// TIA Portal V20 export
DATA_BLOCK "InstCallEquipment"   // DB135
{ DB_Accessible_From_OPC_UA := 'FALSE' }
AUTHOR : ERsystem_FA2_DH. Kim
// stored: AssignedProDiagFB Unit1.Em4.ProDiag, DBAccessibleFromOPCUA false, DBAccessibleFromWebserver false, InstanceOfName Unit1.Em4.CallEquipment, InstanceOfType FB, Namespace Unit1.Em4
"Unit1.Em4.CallEquipment"
   // VAR_INPUT
   //    ZoneOperationEnable { ExternalWritable := 'False'} : "LWONIK_typeSafetyZoneManualOperation";
   // END_VAR
   // VAR_IN_OUT
   //    unitStatus : "LAF_typeUnitStatus";
   //    unitAlarmDB : "LAF_typeAlarms";
   //    emFeedback : "LUC_typeEmFeedback";
   // END_VAR
   // VAR
   //    InstSequenceMainPnP : "Unit1.Em4.Sequence_1_MainPnP";
   //    InstSequenceAlignTable : "Unit1.Em4.Sequence_2_AlignTable";
   //    InstSequenceNgPnP : "Unit1.Em4.Sequence_3_NgPnP";
   //    InstSequenceGaugeRnR : "Unit1.Em4.Sequence_10_GaugeRnR";
   //    instMainPnPHomeJob1 : "LAF_SelectJob";
   //    instMainPnPHomeJob10 : "LAF_SelectJob";
   //    instMainPnPLoadJob2 : "LAF_SelectJob";
   //    instMainPnPUnloadJob3 : "LAF_SelectJob";
   //    instMainPnPAvoidJob4 : "LAF_SelectJob";
   //    instMainPnPOneLoadJob5 : "LAF_SelectJob";
   //    instMainPnPOneUnLoadJob6 : "LAF_SelectJob";
   //    instMainPnPDownWaitJob7 { S7_SetPoint := 'True'} : "LAF_SelectJob";
   //    instAlignTableHomeJob1 : "LAF_SelectJob";
   //    instAlignTableLoadJob2 : "LAF_SelectJob";
   //    instAlignTableVisionJob3 : "LAF_SelectJob";
   //    instAlignTableUnloadJob4 : "LAF_SelectJob";
   //    instAlignTableMotionJob22 : "LAF_SelectJob";
   //    instNgPnPHomeJob1 : "LAF_SelectJob";
   //    instNgPnPLoadJob2 : "LAF_SelectJob";
   //    instNgPnPUnloadJob3 : "LAF_SelectJob";
   //    instGaugeRnRCommonReadyJob1 : "LAF_SelectJob";
   //    instGaugeRnRCommonGetMasterPieceJob2 : "LAF_SelectJob";
   //    instGaugeRnRCommonMainPnPMoveAlignTableStackTableJob3 : "LAF_SelectJob";
   //    instGaugeRnRCommonMainPnp1ToAlignTableJob4 : "LAF_SelectJob";
   //    instGaugeRnRCommonMainPnPMoveReelCutConvyorAlignTableJob5 : "LAF_SelectJob";
   //    instGaugeRnRCommonAlignTableVisionAdjustJob6 : "LAF_SelectJob";
   //    instGaugeRnR1AlignAlignTableToMainPnP1Job10 { S7_SetPoint := 'True'} : "LAF_SelectJob";
   //    instGaugeRnR1AlignMainPnPMoveReelCutConvyorAlignTableJob11 { S7_SetPoint := 'True'} : "LAF_SelectJob";
   //    instGaugeRnR1AlignAlignTableMoveWaitJob12 { S7_SetPoint := 'True'} : "LAF_SelectJob";
   //    instGaugeRnR1AlignUnloadMasterPieceJob13 { S7_SetPoint := 'True'} : "LAF_SelectJob";
   //    instGaugeRnR1StackMainPnPMoveReelCutConvyorAlignTableJob15 { S7_SetPoint := 'True'} : "LAF_SelectJob";
   //    instGaugeRnR1StackAlignTableToMainPnP2Job16 { S7_SetPoint := 'True'} : "LAF_SelectJob";
   //    instGaugeRnR1StackMainPnPMoveAlignTableJob17 { S7_SetPoint := 'True'} : "LAF_SelectJob";
   //    instGaugeRnR1StackAlignTableMoveWaitJob18 { S7_SetPoint := 'True'} : "LAF_SelectJob";
   //    instGaugeRnR1StackMainPnP2ToStackTableJob19 { S7_SetPoint := 'True'} : "LAF_SelectJob";
   //    instGaugeRnR1StackStackTableToMainPnP2Job20 { S7_SetPoint := 'True'} : "LAF_SelectJob";
   //    instGaugeRnR1StackMainPnPMoveReelCutConvyorAlignTableJob21 { S7_SetPoint := 'True'} : "LAF_SelectJob";
   //    instGaugeRnR1StackMainPnP2ToAlignTableJob22 { S7_SetPoint := 'True'} : "LAF_SelectJob";
   //    instGaugeRnR1StackMainPnPMoveAlignTableJob23 { S7_SetPoint := 'True'} : "LAF_SelectJob";
   //    instGaugeRnR1StackAlignTableToMainPnP1Job24 { S7_SetPoint := 'True'} : "LAF_SelectJob";
   //    instGaugeRnR1StackMainPnPMoveReelCutConvyorAlignTableJob25 { S7_SetPoint := 'True'} : "LAF_SelectJob";
   //    instGaugeRnR1StackUnloadMasterPieceJob26 { S7_SetPoint := 'True'} : "LAF_SelectJob";
   //    instGaugeRnR3AlignMainPnPMoveReelCutConvyorAlignTableJob30 { S7_SetPoint := 'True'} : "LAF_SelectJob";
   //    instGaugeRnR3AlignNGPnPLoadMasterPieceJob31 { S7_SetPoint := 'True'} : "LAF_SelectJob";
   //    instGaugeRnR3AlignMainPnP2MoveAlignTableJob32 { S7_SetPoint := 'True'} : "LAF_SelectJob";
   //    instGaugeRnR3AlignAlignTableMoveWaitJob33 { S7_SetPoint := 'True'} : "LAF_SelectJob";
   //    instGaugeRnRCommonCheckCompleteJob39 { S7_SetPoint := 'True'} : "LAF_SelectJob";
   //    instCmPnp1stAnodeDetectSensor { S7_SetPoint := 'True'} : "LBC_DigitalSignalCn";
   //    instCmPnp2ndAnodeDetectSensor { S7_SetPoint := 'True'} : "LBC_DigitalSignalCn";
   //    instCmAnodeAlignTableElectrodeDetectSensor { S7_SetPoint := 'True'} : "LBC_DigitalSignalCn";
   //    instCmAnodeNgBoxFullSensorDetectSensor { S7_SetPoint := 'True'} : "LBC_DigitalSignalCn";
   //    instCmAnodeNgBoxDetectSensor { S7_SetPoint := 'True'} : "LBC_DigitalSignalCn";
   //    instCmAnodeMainPnP1AxisX { S7_SetPoint := 'True'} : "LBC_Axis64Pos_TecPlcCn";
   //    instCmAnodeMainPnP2AxisX { S7_SetPoint := 'True'} : "LBC_Axis64Pos_TecPlcCn";
   //    instCmAnodeMainPnP1AxisY { S7_SetPoint := 'True'} : "LBC_Axis64Pos_TecPlcCn";
   //    instCmAnodeMainPnP1AxisZ { S7_SetPoint := 'True'} : "LBC_Axis64Pos_TecPlcCn";
   //    instCmAnodeMainPnP2AxisZ { S7_SetPoint := 'True'} : "LBC_Axis64Pos_TecPlcCn";
   //    instCmAnodeAlignTableAxisX { S7_SetPoint := 'True'} : "LBC_Axis64Pos_TecPlcCn";
   //    instCmAnodeAlignTableAxisY1 { S7_SetPoint := 'True'} : "LBC_Axis64Pos_TecPlcCn";
   //    instCmAnodeAlignTableAxisY2 { S7_SetPoint := 'True'} : "LBC_Axis64Pos_TecPlcCn";
   //    instInterlockAnodeMainPnP1AxisX { S7_SetPoint := 'True'} : "LER_Axis64Pos_InterlockSummary";
   //    instInterlockAnodeMainPnP1AxisY { S7_SetPoint := 'True'} : "LER_Axis64Pos_InterlockSummary";
   //    instInterlockAnodeMainPnP1AxisZ { S7_SetPoint := 'True'} : "LER_Axis64Pos_InterlockSummary";
   //    instInterlockAnodeMainPnP2AxisX { S7_SetPoint := 'True'} : "LER_Axis64Pos_InterlockSummary";
   //    instInterlockAnodeMainPnP2AxisZ { S7_SetPoint := 'True'} : "LER_Axis64Pos_InterlockSummary";
   //    instInterlockAnodeAlignTableAxisX { S7_SetPoint := 'True'} : "LER_Axis64Pos_InterlockSummary";
   //    instInterlockAnodeAlignTableAxisY1 { S7_SetPoint := 'True'} : "LER_Axis64Pos_InterlockSummary";
   //    instInterlockAnodeAlignTableAxisY2 { S7_SetPoint := 'True'} : "LER_Axis64Pos_InterlockSummary";
   //    instAnodeMainPnP1AxisXSoftCam : "LER_SoftCam_Interface";
   //    instAnodeMainPnP2AxisXSoftCam { S7_SetPoint := 'True'} : "LER_SoftCam_Interface";
   //    instAnodeMainPnP1AxisYSoftCam { S7_SetPoint := 'True'} : "LER_SoftCam_Interface";
   //    instAnodeMainPnP1AxisZSoftCam { S7_SetPoint := 'True'} : "LER_SoftCam_Interface";
   //    instAnodeMainPnP2AxisZSoftCam { S7_SetPoint := 'True'} : "LER_SoftCam_Interface";
   //    instAnodeAlignTableAxisXSoftCam { S7_SetPoint := 'True'} : "LER_SoftCam_Interface";
   //    instAnodeAlignTableAxisY1SoftCam { S7_SetPoint := 'True'} : "LER_SoftCam_Interface";
   //    instAnodeAlignTableAxisY2SoftCam { S7_SetPoint := 'True'} : "LER_SoftCam_Interface";
   //    instCmAnodeMainPnP1RotaryCwCcw { ExternalAccessible := 'False'; ExternalVisible := 'False'; ExternalWritable := 'False'} : "LBC_TwoWayActuatorCn";
   //    instCmAnodeMainPnP1stSuctionPlateVacuum { ExternalAccessible := 'False'; ExternalVisible := 'False'; ExternalWritable := 'False'} : "LBC_TwoWayActuatorCn";
   //    instCmAnodeMainPnP2ndSuctionPlateVacuum { ExternalAccessible := 'False'; ExternalVisible := 'False'; ExternalWritable := 'False'} : "LBC_TwoWayActuatorCn";
   //    instCmAnodeAlignTableSuctionPlateVacuum { ExternalAccessible := 'False'; ExternalVisible := 'False'; ExternalWritable := 'False'; S7_SetPoint := 'True'} : "LBC_TwoWayActuatorCn";
   //    instCmAnodeGlassCleaning { ExternalAccessible := 'False'; ExternalVisible := 'False'; ExternalWritable := 'False'; S7_SetPoint := 'True'} : "LBC_TwoWayActuatorCn";
   //    instCmAnodeNgPnpUpDown { ExternalAccessible := 'False'; ExternalVisible := 'False'; ExternalWritable := 'False'; S7_SetPoint := 'True'} : "LBC_TwoWayActuatorCn";
   //    instCmAnodeNgPnp1stFwdBwd { ExternalAccessible := 'False'; ExternalVisible := 'False'; ExternalWritable := 'False'; S7_SetPoint := 'True'} : "LBC_TwoWayActuatorCn";
   //    instCmAnodeNgPnp2ndFwdBwd { ExternalAccessible := 'False'; ExternalVisible := 'False'; ExternalWritable := 'False'; S7_SetPoint := 'True'} : "LBC_TwoWayActuatorCn";
   //    instCmAnodeMaintenanceMovingFixFwdBwd { ExternalAccessible := 'False'; ExternalVisible := 'False'; ExternalWritable := 'False'; S7_SetPoint := 'True'} : "LBC_TwoWayActuatorCn";
   //    instCmAnodeNgBoxLiftUpDown { ExternalAccessible := 'False'; ExternalVisible := 'False'; ExternalWritable := 'False'; S7_SetPoint := 'True'} : "LBC_TwoWayActuatorCn";
   //    instCmAnodeNgBoxLockUpDown { ExternalAccessible := 'False'; ExternalVisible := 'False'; ExternalWritable := 'False'; S7_SetPoint := 'True'} : "LBC_TwoWayActuatorCn";
   //    instCmAnodeNgPnpVaccum { ExternalAccessible := 'False'; ExternalVisible := 'False'; ExternalWritable := 'False'; S7_SetPoint := 'True'} : "LBC_TwoWayActuatorCn";
   //    instCmAnodeConveyorCoverFwdBwd { S7_SetPoint := 'True'} : "LBC_TwoWayActuatorCn";
   //    instCmAnodeConveyorPickUpBlower { S7_SetPoint := 'True'} : "LBC_TwoWayActuatorCn";
   //    instCmAnodeVisionControllerInterface { ExternalAccessible := 'False'; ExternalVisible := 'False'; ExternalWritable := 'False'; S7_SetPoint := 'True'} : "LER_Vision_XGX2000";
   //    instAlignVisionConversion : "LER_AlignVisionConversion";
   //    instManageAlarms { ExternalWritable := 'False'} : "LAF_ManageAlarms";
   //    instLER_BrakeTestAnodeMainPnP1AxisZ : "LER_BrakeTest";
   //    instLER_BrakeTestAnodeMainPnP2AxisZ { S7_SetPoint := 'True'} : "LER_BrakeTest";
   //    instEventsPFE : "Unit1.Em4.EventsPFE";
   //    statUnitStatus { ExternalWritable := 'False'} : "LAF_typeUnitStatus";
   //    statSlmStatus { ExternalWritable := 'False'} : Struct
   //       running : Bool;
   //       powerOff : Bool;
   //    END_STRUCT;
   //    statAllBrakeTest { ExternalWritable := 'False'} : "LER_typeBrakeTestUnitCommands";
   //    statInterlockTonTime { ExternalAccessible := 'False'; ExternalVisible := 'False'; ExternalWritable := 'False'} : Struct
   //       mainPnP1AxisX : Array[0..15] of TON_TIME;
   //       mainPnP1AxisY : Array[0..15] of TON_TIME;
   //       mainPnP1AxisZ : Array[0..15] of TON_TIME;
   //       mainPnP2AxisX : Array[0..15] of TON_TIME;
   //       mainPnP2AxisZ : Array[0..15] of TON_TIME;
   //       alignTableAxisX : Array[0..15] of TON_TIME;
   //       alignTableAxisY1 : Array[0..15] of TON_TIME;
   //       alignTableAxisY2 : Array[0..15] of TON_TIME;
   //    END_STRUCT;
   //    statTonTime { ExternalAccessible := 'False'; ExternalVisible := 'False'; ExternalWritable := 'False'} : Array[0..1999] of TON_TIME;
   //    statTofTime { ExternalAccessible := 'False'; ExternalVisible := 'False'; ExternalWritable := 'False'} : Array[0..99] of TOF_TIME;
   //    statPulse { ExternalAccessible := 'False'; ExternalVisible := 'False'; ExternalWritable := 'False'} : Struct
   //       miscellaneous : Array[0..99] of Bool;
   //       workingDone : Struct
   //          mainPnP : Array[0..99] of Bool;
   //          alignTable : Array[0..99] of Bool;
   //          ngPnP : Array[0..99] of Bool;
   //       END_STRUCT;
   //       axisEnable : Array[0..99] of Bool;
   //       brakeTest : Array[0..99] of Bool;
   //    END_STRUCT;
   //    statEnableManualCmds : Bool := TRUE;
   //    Scan_on : Bool;
   //    "*** Interlock Axis ***" { ExternalAccessible := 'False'; ExternalVisible := 'False'; ExternalWritable := 'False'} : Bool;
   //    "AnodeMainPnP1AxisX Home" { S7_SetPoint := 'True'} : "Homing.LER_Axis";
   //    "AnodeMainPnP1AxisX Jog_CW" { S7_SetPoint := 'True'} : "Jog.LER_Axis";
   //    "AnodeMainPnP1AxisX Jog_CCW" { S7_SetPoint := 'True'} : "Jog.LER_Axis";
   //    "AnodeMainPnP1AxisX Position_" { S7_SetPoint := 'True'} : Array[0..5] of "Position.LER_Axis";
   //    "AnodeMainPnP2AxisX Home" { S7_SetPoint := 'True'} : "Homing.LER_Axis";
   //    "AnodeMainPnP2AxisX Jog_CW" { S7_SetPoint := 'True'} : "Jog.LER_Axis";
   //    "AnodeMainPnP2AxisX Jog_CCW" { S7_SetPoint := 'True'} : "Jog.LER_Axis";
   //    "AnodeMainPnP2AxisX Position_" { S7_SetPoint := 'True'} : Array[0..5] of "Position.LER_Axis";
   //    "AnodeMainPnP1AxisY Home" { S7_SetPoint := 'True'} : "Homing.LER_Axis";
   //    "AnodeMainPnP1AxisY Jog_CW" { S7_SetPoint := 'True'} : "Jog.LER_Axis";
   //    "AnodeMainPnP1AxisY Jog_CCW" { S7_SetPoint := 'True'} : "Jog.LER_Axis";
   //    "AnodeMainPnP1AxisY Position_" { S7_SetPoint := 'True'} : Array[0..5] of "Position.LER_Axis";
   //    "AnodeMainPnP1AxisZ Home" { S7_SetPoint := 'True'} : "Homing.LER_Axis";
   //    "AnodeMainPnP1AxisZ Jog_CW" { S7_SetPoint := 'True'} : "Jog.LER_Axis";
   //    "AnodeMainPnP1AxisZ Jog_CCW" { S7_SetPoint := 'True'} : "Jog.LER_Axis";
   //    "AnodeMainPnP1AxisZ Position_" { S7_SetPoint := 'True'} : Array[0..5] of "Position.LER_Axis";
   //    "AnodeMainPnP2AxisZ Home" { S7_SetPoint := 'True'} : "Homing.LER_Axis";
   //    "AnodeMainPnP2AxisZ Jog_CW" { S7_SetPoint := 'True'} : "Jog.LER_Axis";
   //    "AnodeMainPnP2AxisZ Jog_CCW" { S7_SetPoint := 'True'} : "Jog.LER_Axis";
   //    "AnodeMainPnP2AxisZ Position_" { S7_SetPoint := 'True'} : Array[0..5] of "Position.LER_Axis";
   //    "AnodeAlignTableAxisX Home" { S7_SetPoint := 'True'} : "Homing.LER_Axis";
   //    "AnodeAlignTableAxisX Jog_CW" { S7_SetPoint := 'True'} : "Jog.LER_Axis";
   //    "AnodeAlignTableAxisX Jog_CCW" { S7_SetPoint := 'True'} : "Jog.LER_Axis";
   //    "AnodeAlignTableAxisX Position_" { S7_SetPoint := 'True'} : Array[0..5] of "Position.LER_Axis";
   //    "AnodeAlignTableAxisY1 Home" { S7_SetPoint := 'True'} : "Homing.LER_Axis";
   //    "AnodeAlignTableAxisY1 Jog_CW" { S7_SetPoint := 'True'} : "Jog.LER_Axis";
   //    "AnodeAlignTableAxisY1 Jog_CCW" { S7_SetPoint := 'True'} : "Jog.LER_Axis";
   //    "AnodeAlignTableAxisY1 Position_" { S7_SetPoint := 'True'} : Array[0..5] of "Position.LER_Axis";
   //    "AnodeAlignTableAxisY2 Home" { S7_SetPoint := 'True'} : "Homing.LER_Axis";
   //    "AnodeAlignTableAxisY2 Jog_CW" { S7_SetPoint := 'True'} : "Jog.LER_Axis";
   //    "AnodeAlignTableAxisY2 Jog_CCW" { S7_SetPoint := 'True'} : "Jog.LER_Axis";
   //    "AnodeAlignTableAxisY2 Position_" { S7_SetPoint := 'True'} : Array[0..5] of "Position.LER_Axis";
   //    "*** Interlock Actuator ******" { ExternalAccessible := 'False'; ExternalVisible := 'False'; ExternalWritable := 'False'} : Bool;
   //    "AnodeNgBoxLiftUpDown Home" { S7_SetPoint := 'True'} : "Cylinder.LER_Actuator";
   //    "AnodeNgBoxLiftUpDown Work" { S7_SetPoint := 'True'} : "Cylinder.LER_Actuator";
   //    "AnodeNgBoxLockUpDown Home" { S7_SetPoint := 'True'} : "Cylinder.LER_Actuator";
   //    "AnodeNgBoxLockUpDown Work" { S7_SetPoint := 'True'} : "Cylinder.LER_Actuator";
   //    "AnodeMaintenanceMovingFixFrontFwdBwd Home" { S7_SetPoint := 'True'} : "Cylinder.LER_Actuator";
   //    "AnodeMaintenanceMovingFixFrontFwdBwd Work" { S7_SetPoint := 'True'} : "Cylinder.LER_Actuator";
   //    "AnodeGlassCleaning Home" { S7_SetPoint := 'True'} : "Cylinder.LER_Actuator";
   //    "AnodeGlassCleaning Work" { S7_SetPoint := 'True'} : "Cylinder.LER_Actuator";
   //    "AnodeNgPnp1stFwdBwd Home" { S7_SetPoint := 'True'} : "Cylinder.LER_Actuator";
   //    "AnodeNgPnp1stFwdBwd Work" { S7_SetPoint := 'True'} : "Cylinder.LER_Actuator";
   //    "AnodeNgPnpUpDown Home" { S7_SetPoint := 'True'} : "Cylinder.LER_Actuator";
   //    "AnodeNgPnpUpDown Work" { S7_SetPoint := 'True'} : "Cylinder.LER_Actuator";
   //    "AnodeMainPnP1RotaryCwCcw Home" { S7_SetPoint := 'True'} : "Cylinder.LER_Actuator";
   //    "AnodeMainPnP1RotaryCwCcw Work" { S7_SetPoint := 'True'} : "Cylinder.LER_Actuator";
   //    "AnodeNgPnp2ndFwdBwd Home" { S7_SetPoint := 'True'} : "Cylinder.LER_Actuator";
   //    "AnodeNgPnp2ndFwdBwd Work" { S7_SetPoint := 'True'} : "Cylinder.LER_Actuator";
   //    Tracking_04 { S7_SetPoint := 'True'} : "Unit1.Em4.PartData";
   //    AXIS5 : "LER_CM_Name";
   //    AXIS11 : "LER_CM_Name";
   //    AXIS14 : "LER_CM_Name";
   //    Cylinder13 : "LER_CM_Name";
   //    Cylinder18 : "LER_CM_Name";
   //    Vaccum10 : "LER_CM_Name";
   //    instAlignVisionHistory { S7_SetPoint := 'True'} : "LER_visionHistory";
   //    instAlignMoveCalibration { S7_SetPoint := 'True'} : "LER_AlignMoveCalibration";
   //    instAlignThetaCalibration { S7_SetPoint := 'True'} : "LER_AlignThetaCalibration";
   //    instAlignSyncMove { S7_SetPoint := 'True'} : "LER_AlignSyncMove";
   //    citi_Ptrig : Array[0..20] of Bool;
   //    citiTon : Array[0..20] of TON_TIME;
   //    citi : Time;
   //    citiTest : Array[0..20] of Bool;
   // END_VAR
BEGIN
   ZoneOperationEnable.autoStartEnable := FALSE;
   ZoneOperationEnable.doorLockEnable := TRUE;
   ZoneOperationEnable.doorUnlockEnable := TRUE;
   ZoneOperationEnable.rc_AutoEnable := FALSE;
   ZoneOperationEnable.rc_RollChangeEnable := FALSE;
   ZoneOperationEnable.rc_DoorLockEnable := TRUE;
   ZoneOperationEnable.rc_DoorUnlockEnable := TRUE;
   ZoneOperationEnable.hmiOperationEnable := TRUE;
   ZoneOperationEnable.phmiOperationEnable := FALSE;
   instCmPnp1stAnodeDetectSensor.enable := TRUE;
   instCmPnp1stAnodeDetectSensor.parentReferenceDesignator := WSTRING#'';
   instCmPnp1stAnodeDetectSensor.digitalValue := FALSE;
   instCmPnp1stAnodeDetectSensor.simulatedDigitalValue := FALSE;
   instCmPnp1stAnodeDetectSensor.statProcessValues.enable := TRUE;
   instCmPnp1stAnodeDetectSensor.statProcessValues.referenceDesignator := WSTRING#'Pnp1stAnodeDetect';
   instCmPnp1stAnodeDetectSensor.statProcessValues.simulation := FALSE;
   instCmPnp1stAnodeDetectSensor.statProcessValues.processValue := FALSE;
   instCmPnp1stAnodeDetectSensor.statProcessValues.error := FALSE;
   instCmPnp1stAnodeDetectSensor.statProcessValues.status := 16#0000;
   instCmPnp1stAnodeDetectSensor.statDiagnostics.status := 16#0000;
   instCmPnp1stAnodeDetectSensor.statDiagnostics.subfunctionStatus := 16#0000;
   instCmPnp1stAnodeDetectSensor.statDiagnostics.stateNumber := 0;
   instCmPnp1stAnodeDetectSensor.statEmptyDiagnostics.status := 16#0000;
   instCmPnp1stAnodeDetectSensor.statEmptyDiagnostics.subfunctionStatus := 16#0000;
   instCmPnp1stAnodeDetectSensor.statEmptyDiagnostics.stateNumber := 0;
   instCmPnp1stAnodeDetectSensor.instOnDelay.PT := T#0MS;
   instCmPnp1stAnodeDetectSensor.instOnDelay.IN := FALSE;
   instCmPnp1stAnodeDetectSensor.instOffDelay.PT := T#0MS;
   instCmPnp1stAnodeDetectSensor.instOffDelay.IN := FALSE;
   instCmPnp1stAnodeDetectSensor.statDisableAlarms := FALSE;
   instCmPnp1stAnodeDetectSensor.statErrorState := 16#0000;
   instCmPnp1stAnodeDetectSensor.statFirstCall := FALSE;
   instCmPnp1stAnodeDetectSensor.statResetPrevious := FALSE;
   instCmPnp1stAnodeDetectSensor.statEnablePrevious := TRUE;
   instCmPnp1stAnodeDetectSensor.statProcessValuePrevious := FALSE;
   instCmPnp2ndAnodeDetectSensor.enable := TRUE;
   instCmPnp2ndAnodeDetectSensor.parentReferenceDesignator := WSTRING#'';
   instCmPnp2ndAnodeDetectSensor.digitalValue := FALSE;
   instCmPnp2ndAnodeDetectSensor.simulatedDigitalValue := FALSE;
   instCmPnp2ndAnodeDetectSensor.statProcessValues.enable := TRUE;
   instCmPnp2ndAnodeDetectSensor.statProcessValues.referenceDesignator := WSTRING#'Pnp2ndAnodeDetect';
   instCmPnp2ndAnodeDetectSensor.statProcessValues.simulation := FALSE;
   instCmPnp2ndAnodeDetectSensor.statProcessValues.processValue := FALSE;
   instCmPnp2ndAnodeDetectSensor.statProcessValues.error := FALSE;
   instCmPnp2ndAnodeDetectSensor.statProcessValues.status := 16#0000;
   instCmPnp2ndAnodeDetectSensor.statDiagnostics.status := 16#0000;
   instCmPnp2ndAnodeDetectSensor.statDiagnostics.subfunctionStatus := 16#0000;
   instCmPnp2ndAnodeDetectSensor.statDiagnostics.stateNumber := 0;
   instCmPnp2ndAnodeDetectSensor.statEmptyDiagnostics.status := 16#0000;
   instCmPnp2ndAnodeDetectSensor.statEmptyDiagnostics.subfunctionStatus := 16#0000;
   instCmPnp2ndAnodeDetectSensor.statEmptyDiagnostics.stateNumber := 0;
   instCmPnp2ndAnodeDetectSensor.instOnDelay.PT := T#0MS;
   instCmPnp2ndAnodeDetectSensor.instOnDelay.IN := FALSE;
   instCmPnp2ndAnodeDetectSensor.instOffDelay.PT := T#0MS;
   instCmPnp2ndAnodeDetectSensor.instOffDelay.IN := FALSE;
   instCmPnp2ndAnodeDetectSensor.statDisableAlarms := FALSE;
   instCmPnp2ndAnodeDetectSensor.statErrorState := 16#0000;
   instCmPnp2ndAnodeDetectSensor.statFirstCall := FALSE;
   instCmPnp2ndAnodeDetectSensor.statResetPrevious := FALSE;
   instCmPnp2ndAnodeDetectSensor.statEnablePrevious := TRUE;
   instCmPnp2ndAnodeDetectSensor.statProcessValuePrevious := FALSE;
   instCmAnodeAlignTableElectrodeDetectSensor.enable := TRUE;
   instCmAnodeAlignTableElectrodeDetectSensor.parentReferenceDesignator := WSTRING#'';
   instCmAnodeAlignTableElectrodeDetectSensor.digitalValue := FALSE;
   instCmAnodeAlignTableElectrodeDetectSensor.simulatedDigitalValue := FALSE;
   instCmAnodeAlignTableElectrodeDetectSensor.statProcessValues.enable := TRUE;
   instCmAnodeAlignTableElectrodeDetectSensor.statProcessValues.referenceDesignator := WSTRING#'AlignTableElectrodeDetect';
   instCmAnodeAlignTableElectrodeDetectSensor.statProcessValues.simulation := FALSE;
   instCmAnodeAlignTableElectrodeDetectSensor.statProcessValues.processValue := FALSE;
   instCmAnodeAlignTableElectrodeDetectSensor.statProcessValues.error := FALSE;
   instCmAnodeAlignTableElectrodeDetectSensor.statProcessValues.status := 16#0000;
   instCmAnodeAlignTableElectrodeDetectSensor.statDiagnostics.status := 16#0000;
   instCmAnodeAlignTableElectrodeDetectSensor.statDiagnostics.subfunctionStatus := 16#0000;
   instCmAnodeAlignTableElectrodeDetectSensor.statDiagnostics.stateNumber := 0;
   instCmAnodeAlignTableElectrodeDetectSensor.statEmptyDiagnostics.status := 16#0000;
   instCmAnodeAlignTableElectrodeDetectSensor.statEmptyDiagnostics.subfunctionStatus := 16#0000;
   instCmAnodeAlignTableElectrodeDetectSensor.statEmptyDiagnostics.stateNumber := 0;
   instCmAnodeAlignTableElectrodeDetectSensor.instOnDelay.PT := T#0MS;
   instCmAnodeAlignTableElectrodeDetectSensor.instOnDelay.IN := FALSE;
   instCmAnodeAlignTableElectrodeDetectSensor.instOffDelay.PT := T#0MS;
   instCmAnodeAlignTableElectrodeDetectSensor.instOffDelay.IN := FALSE;
   instCmAnodeAlignTableElectrodeDetectSensor.statDisableAlarms := FALSE;
   instCmAnodeAlignTableElectrodeDetectSensor.statErrorState := 16#0000;
   instCmAnodeAlignTableElectrodeDetectSensor.statFirstCall := FALSE;
   instCmAnodeAlignTableElectrodeDetectSensor.statResetPrevious := FALSE;
   instCmAnodeAlignTableElectrodeDetectSensor.statEnablePrevious := TRUE;
   instCmAnodeAlignTableElectrodeDetectSensor.statProcessValuePrevious := FALSE;
   instCmAnodeNgBoxFullSensorDetectSensor.enable := TRUE;
   instCmAnodeNgBoxFullSensorDetectSensor.parentReferenceDesignator := WSTRING#'';
   instCmAnodeNgBoxFullSensorDetectSensor.digitalValue := TRUE;
   instCmAnodeNgBoxFullSensorDetectSensor.simulatedDigitalValue := FALSE;
   instCmAnodeNgBoxFullSensorDetectSensor.statProcessValues.enable := TRUE;
   instCmAnodeNgBoxFullSensorDetectSensor.statProcessValues.referenceDesignator := WSTRING#'NgBoxFullSensorDetect';
   instCmAnodeNgBoxFullSensorDetectSensor.statProcessValues.simulation := FALSE;
   instCmAnodeNgBoxFullSensorDetectSensor.statProcessValues.processValue := TRUE;
   instCmAnodeNgBoxFullSensorDetectSensor.statProcessValues.error := FALSE;
   instCmAnodeNgBoxFullSensorDetectSensor.statProcessValues.status := 16#0000;
   instCmAnodeNgBoxFullSensorDetectSensor.statDiagnostics.status := 16#0000;
   instCmAnodeNgBoxFullSensorDetectSensor.statDiagnostics.subfunctionStatus := 16#0000;
   instCmAnodeNgBoxFullSensorDetectSensor.statDiagnostics.stateNumber := 0;
   instCmAnodeNgBoxFullSensorDetectSensor.statEmptyDiagnostics.status := 16#0000;
   instCmAnodeNgBoxFullSensorDetectSensor.statEmptyDiagnostics.subfunctionStatus := 16#0000;
   instCmAnodeNgBoxFullSensorDetectSensor.statEmptyDiagnostics.stateNumber := 0;
   instCmAnodeNgBoxFullSensorDetectSensor.instOnDelay.PT := T#0MS;
   instCmAnodeNgBoxFullSensorDetectSensor.instOnDelay.IN := FALSE;
   instCmAnodeNgBoxFullSensorDetectSensor.instOffDelay.PT := T#0MS;
   instCmAnodeNgBoxFullSensorDetectSensor.instOffDelay.IN := FALSE;
   instCmAnodeNgBoxFullSensorDetectSensor.statDisableAlarms := FALSE;
   instCmAnodeNgBoxFullSensorDetectSensor.statErrorState := 16#0000;
   instCmAnodeNgBoxFullSensorDetectSensor.statFirstCall := FALSE;
   instCmAnodeNgBoxFullSensorDetectSensor.statResetPrevious := FALSE;
   instCmAnodeNgBoxFullSensorDetectSensor.statEnablePrevious := TRUE;
   instCmAnodeNgBoxFullSensorDetectSensor.statProcessValuePrevious := TRUE;
   instCmAnodeNgBoxDetectSensor.enable := TRUE;
   instCmAnodeNgBoxDetectSensor.parentReferenceDesignator := WSTRING#'';
   instCmAnodeNgBoxDetectSensor.digitalValue := TRUE;
   instCmAnodeNgBoxDetectSensor.simulatedDigitalValue := FALSE;
   instCmAnodeNgBoxDetectSensor.statProcessValues.enable := TRUE;
   instCmAnodeNgBoxDetectSensor.statProcessValues.referenceDesignator := WSTRING#'NgBoxDetect';
   instCmAnodeNgBoxDetectSensor.statProcessValues.simulation := FALSE;
   instCmAnodeNgBoxDetectSensor.statProcessValues.processValue := TRUE;
   instCmAnodeNgBoxDetectSensor.statProcessValues.error := FALSE;
   instCmAnodeNgBoxDetectSensor.statProcessValues.status := 16#0000;
   instCmAnodeNgBoxDetectSensor.statDiagnostics.status := 16#0000;
   instCmAnodeNgBoxDetectSensor.statDiagnostics.subfunctionStatus := 16#0000;
   instCmAnodeNgBoxDetectSensor.statDiagnostics.stateNumber := 0;
   instCmAnodeNgBoxDetectSensor.statEmptyDiagnostics.status := 16#0000;
   instCmAnodeNgBoxDetectSensor.statEmptyDiagnostics.subfunctionStatus := 16#0000;
   instCmAnodeNgBoxDetectSensor.statEmptyDiagnostics.stateNumber := 0;
   instCmAnodeNgBoxDetectSensor.instOnDelay.PT := T#0MS;
   instCmAnodeNgBoxDetectSensor.instOnDelay.IN := FALSE;
   instCmAnodeNgBoxDetectSensor.instOffDelay.PT := T#0MS;
   instCmAnodeNgBoxDetectSensor.instOffDelay.IN := FALSE;
   instCmAnodeNgBoxDetectSensor.statDisableAlarms := FALSE;
   instCmAnodeNgBoxDetectSensor.statErrorState := 16#0000;
   instCmAnodeNgBoxDetectSensor.statFirstCall := FALSE;
   instCmAnodeNgBoxDetectSensor.statResetPrevious := FALSE;
   instCmAnodeNgBoxDetectSensor.statEnablePrevious := TRUE;
   instCmAnodeNgBoxDetectSensor.statProcessValuePrevious := TRUE;
   instCmAnodeMainPnP1RotaryCwCcw.enable := TRUE;
   instCmAnodeMainPnP1RotaryCwCcw.parentReferenceDesignator := WSTRING#'';
   instCmAnodeMainPnP1RotaryCwCcw.feedbackHomePos := FALSE;
   instCmAnodeMainPnP1RotaryCwCcw.feedbackWorkPos := TRUE;
   instCmAnodeMainPnP1RotaryCwCcw.enableManualCmds := TRUE;
   instCmAnodeMainPnP1RotaryCwCcw.interlockWorkPos := FALSE;
   instCmAnodeMainPnP1RotaryCwCcw.interlockHomePos := FALSE;
   instCmAnodeMainPnP1RotaryCwCcw.goToHomePos := FALSE;
   instCmAnodeMainPnP1RotaryCwCcw.goToWorkPos := FALSE;
   instCmAnodeMainPnP1RotaryCwCcw.statProcessValues.enable := TRUE;
   instCmAnodeMainPnP1RotaryCwCcw.statProcessValues.referenceDesignator := WSTRING#'MainPnP1RotaryCwCcw';
   instCmAnodeMainPnP1RotaryCwCcw.statProcessValues.commandHomePos := FALSE;
   instCmAnodeMainPnP1RotaryCwCcw.statProcessValues.commandWorkPos := FALSE;
   instCmAnodeMainPnP1RotaryCwCcw.statProcessValues.goToHomePos := FALSE;
   instCmAnodeMainPnP1RotaryCwCcw.statProcessValues.goToWorkPos := FALSE;
   instCmAnodeMainPnP1RotaryCwCcw.statProcessValues.inHomePos := FALSE;
   instCmAnodeMainPnP1RotaryCwCcw.statProcessValues.inWorkPos := FALSE;
   instCmAnodeMainPnP1RotaryCwCcw.statProcessValues.reset := FALSE;
   instCmAnodeMainPnP1RotaryCwCcw.statProcessValues.enableManualCmds := TRUE;
   instCmAnodeMainPnP1RotaryCwCcw.statProcessValues.error := FALSE;
   instCmAnodeMainPnP1RotaryCwCcw.statProcessValues.interlockHomePos := FALSE;
   instCmAnodeMainPnP1RotaryCwCcw.statProcessValues.interlockWorkPos := FALSE;
   instCmAnodeMainPnP1RotaryCwCcw.statProcessValues.status := 16#7100;
   instCmAnodeMainPnP1RotaryCwCcw.statProcessValues.interlockWarningWorkPos := FALSE;
   instCmAnodeMainPnP1RotaryCwCcw.statProcessValues.interlockWarningHomePos := FALSE;
   instCmAnodeMainPnP1RotaryCwCcw.statCurrentInputs.commandHomePos := FALSE;
   instCmAnodeMainPnP1RotaryCwCcw.statCurrentInputs.commandWorkPos := FALSE;
   instCmAnodeMainPnP1RotaryCwCcw.statCurrentInputs.reset := FALSE;
   instCmAnodeMainPnP1RotaryCwCcw.statPreviousInputs.commandHomePos := FALSE;
   instCmAnodeMainPnP1RotaryCwCcw.statPreviousInputs.commandWorkPos := FALSE;
   instCmAnodeMainPnP1RotaryCwCcw.statPreviousInputs.reset := FALSE;
   instCmAnodeMainPnP1RotaryCwCcw.statCurrentInterface.commandHomePos := FALSE;
   instCmAnodeMainPnP1RotaryCwCcw.statCurrentInterface.commandWorkPos := FALSE;
   instCmAnodeMainPnP1RotaryCwCcw.statCurrentInterface.reset := FALSE;
   instCmAnodeMainPnP1RotaryCwCcw.statPreviousInterface.commandHomePos := FALSE;
   instCmAnodeMainPnP1RotaryCwCcw.statPreviousInterface.commandWorkPos := FALSE;
   instCmAnodeMainPnP1RotaryCwCcw.statPreviousInterface.reset := FALSE;
   instCmAnodeMainPnP1RotaryCwCcw.statEmptyDiagnostics.status := 16#0000;
   instCmAnodeMainPnP1RotaryCwCcw.statEmptyDiagnostics.subfunctionStatus := 16#0000;
   instCmAnodeMainPnP1RotaryCwCcw.statEmptyDiagnostics.stateNumber := 0;
   instCmAnodeMainPnP1RotaryCwCcw.instTimerReachPos.PT := T#0MS;
   instCmAnodeMainPnP1RotaryCwCcw.instTimerReachPos.IN := FALSE;
   instCmAnodeMainPnP1RotaryCwCcw.instTimerLeavePos.PT := T#0MS;
   instCmAnodeMainPnP1RotaryCwCcw.instTimerLeavePos.IN := FALSE;
   instCmAnodeMainPnP1RotaryCwCcw.instTimerDiscrepancyCheck.PT := T#0MS;
   instCmAnodeMainPnP1RotaryCwCcw.instTimerDiscrepancyCheck.IN := FALSE;
   instCmAnodeMainPnP1RotaryCwCcw.statDisableAlarms := TRUE;
   instCmAnodeMainPnP1RotaryCwCcw.statDiagnostics.status := 16#7003;
   instCmAnodeMainPnP1RotaryCwCcw.statDiagnostics.subfunctionStatus := 16#0000;
   instCmAnodeMainPnP1RotaryCwCcw.statDiagnostics.stateNumber := 0;
   instCmAnodeMainPnP1RotaryCwCcw.statEnablePrevious := TRUE;
   instCmAnodeMainPnP1RotaryCwCcw.statFirstCall := FALSE;
   instCmAnodeMainPnP1RotaryCwCcw.statResetPrevious := FALSE;
   instCmAnodeMainPnP1RotaryCwCcw.statValid := TRUE;
   instCmAnodeMainPnP1RotaryCwCcw.statBusy := TRUE;
   instCmAnodeMainPnP1RotaryCwCcw.statError := FALSE;
   instCmAnodeMainPnP1RotaryCwCcw.statInterlockWorkOff := FALSE;
   instCmAnodeMainPnP1RotaryCwCcw.statInterlockHomeOff := FALSE;
   instCmAnodeMainPnP1RotaryCwCcw.statFbState := 50;
   instCmAnodeMainPnP1RotaryCwCcw.statFbStatePrevious := 50;
   instCmAnodeMainPnP1RotaryCwCcw.statErrorUserCleared := FALSE;
   instCmAnodeMainPnP1RotaryCwCcw.statErrorAutoCleared := FALSE;
   instCmAnodeMainPnP1RotaryCwCcw.statErrorState := 16#0000;
   instCmAnodeMainPnP1RotaryCwCcw.statDisablingCompleted := FALSE;
   instCmAnodeMainPnP1RotaryCwCcw.statFeedbackHomePos := FALSE;
   instCmAnodeMainPnP1RotaryCwCcw.statFeedbackWorkPos := TRUE;
   instCmAnodeMainPnP1stSuctionPlateVacuum.enable := TRUE;
   instCmAnodeMainPnP1stSuctionPlateVacuum.parentReferenceDesignator := WSTRING#'';
   instCmAnodeMainPnP1stSuctionPlateVacuum.feedbackHomePos := TRUE;
   instCmAnodeMainPnP1stSuctionPlateVacuum.feedbackWorkPos := FALSE;
   instCmAnodeMainPnP1stSuctionPlateVacuum.enableManualCmds := TRUE;
   instCmAnodeMainPnP1stSuctionPlateVacuum.interlockWorkPos := TRUE;
   instCmAnodeMainPnP1stSuctionPlateVacuum.interlockHomePos := TRUE;
   instCmAnodeMainPnP1stSuctionPlateVacuum.goToHomePos := FALSE;
   instCmAnodeMainPnP1stSuctionPlateVacuum.goToWorkPos := FALSE;
   instCmAnodeMainPnP1stSuctionPlateVacuum.statProcessValues.enable := TRUE;
   instCmAnodeMainPnP1stSuctionPlateVacuum.statProcessValues.referenceDesignator := WSTRING#'MainPnP1Vacuum';
   instCmAnodeMainPnP1stSuctionPlateVacuum.statProcessValues.commandHomePos := FALSE;
   instCmAnodeMainPnP1stSuctionPlateVacuum.statProcessValues.commandWorkPos := FALSE;
   instCmAnodeMainPnP1stSuctionPlateVacuum.statProcessValues.goToHomePos := FALSE;
   instCmAnodeMainPnP1stSuctionPlateVacuum.statProcessValues.goToWorkPos := FALSE;
   instCmAnodeMainPnP1stSuctionPlateVacuum.statProcessValues.inHomePos := TRUE;
   instCmAnodeMainPnP1stSuctionPlateVacuum.statProcessValues.inWorkPos := FALSE;
   instCmAnodeMainPnP1stSuctionPlateVacuum.statProcessValues.reset := FALSE;
   instCmAnodeMainPnP1stSuctionPlateVacuum.statProcessValues.enableManualCmds := TRUE;
   instCmAnodeMainPnP1stSuctionPlateVacuum.statProcessValues.error := FALSE;
   instCmAnodeMainPnP1stSuctionPlateVacuum.statProcessValues.interlockHomePos := TRUE;
   instCmAnodeMainPnP1stSuctionPlateVacuum.statProcessValues.interlockWorkPos := TRUE;
   instCmAnodeMainPnP1stSuctionPlateVacuum.statProcessValues.status := 16#7003;
   instCmAnodeMainPnP1stSuctionPlateVacuum.statProcessValues.interlockWarningWorkPos := FALSE;
   instCmAnodeMainPnP1stSuctionPlateVacuum.statProcessValues.interlockWarningHomePos := FALSE;
   instCmAnodeMainPnP1stSuctionPlateVacuum.statCurrentInputs.commandHomePos := FALSE;
   instCmAnodeMainPnP1stSuctionPlateVacuum.statCurrentInputs.commandWorkPos := FALSE;
   instCmAnodeMainPnP1stSuctionPlateVacuum.statCurrentInputs.reset := FALSE;
   instCmAnodeMainPnP1stSuctionPlateVacuum.statPreviousInputs.commandHomePos := FALSE;
   instCmAnodeMainPnP1stSuctionPlateVacuum.statPreviousInputs.commandWorkPos := FALSE;
   instCmAnodeMainPnP1stSuctionPlateVacuum.statPreviousInputs.reset := FALSE;
   instCmAnodeMainPnP1stSuctionPlateVacuum.statCurrentInterface.commandHomePos := FALSE;
   instCmAnodeMainPnP1stSuctionPlateVacuum.statCurrentInterface.commandWorkPos := FALSE;
   instCmAnodeMainPnP1stSuctionPlateVacuum.statCurrentInterface.reset := FALSE;
   instCmAnodeMainPnP1stSuctionPlateVacuum.statPreviousInterface.commandHomePos := FALSE;
   instCmAnodeMainPnP1stSuctionPlateVacuum.statPreviousInterface.commandWorkPos := FALSE;
   instCmAnodeMainPnP1stSuctionPlateVacuum.statPreviousInterface.reset := FALSE;
   instCmAnodeMainPnP1stSuctionPlateVacuum.statEmptyDiagnostics.status := 16#0000;
   instCmAnodeMainPnP1stSuctionPlateVacuum.statEmptyDiagnostics.subfunctionStatus := 16#0000;
   instCmAnodeMainPnP1stSuctionPlateVacuum.statEmptyDiagnostics.stateNumber := 0;
   instCmAnodeMainPnP1stSuctionPlateVacuum.instTimerReachPos.PT := T#0MS;
   instCmAnodeMainPnP1stSuctionPlateVacuum.instTimerReachPos.IN := FALSE;
   instCmAnodeMainPnP1stSuctionPlateVacuum.instTimerLeavePos.PT := T#0MS;
   instCmAnodeMainPnP1stSuctionPlateVacuum.instTimerLeavePos.IN := FALSE;
   instCmAnodeMainPnP1stSuctionPlateVacuum.instTimerDiscrepancyCheck.PT := T#0MS;
   instCmAnodeMainPnP1stSuctionPlateVacuum.instTimerDiscrepancyCheck.IN := FALSE;
   instCmAnodeMainPnP1stSuctionPlateVacuum.statDisableAlarms := FALSE;
   instCmAnodeMainPnP1stSuctionPlateVacuum.statDiagnostics.status := 16#7003;
   instCmAnodeMainPnP1stSuctionPlateVacuum.statDiagnostics.subfunctionStatus := 16#0000;
   instCmAnodeMainPnP1stSuctionPlateVacuum.statDiagnostics.stateNumber := 0;
   instCmAnodeMainPnP1stSuctionPlateVacuum.statEnablePrevious := TRUE;
   instCmAnodeMainPnP1stSuctionPlateVacuum.statFirstCall := FALSE;
   instCmAnodeMainPnP1stSuctionPlateVacuum.statResetPrevious := FALSE;
   instCmAnodeMainPnP1stSuctionPlateVacuum.statValid := TRUE;
   instCmAnodeMainPnP1stSuctionPlateVacuum.statBusy := TRUE;
   instCmAnodeMainPnP1stSuctionPlateVacuum.statError := FALSE;
   instCmAnodeMainPnP1stSuctionPlateVacuum.statInterlockWorkOff := FALSE;
   instCmAnodeMainPnP1stSuctionPlateVacuum.statInterlockHomeOff := FALSE;
   instCmAnodeMainPnP1stSuctionPlateVacuum.statFbState := 50;
   instCmAnodeMainPnP1stSuctionPlateVacuum.statFbStatePrevious := 50;
   instCmAnodeMainPnP1stSuctionPlateVacuum.statErrorUserCleared := FALSE;
   instCmAnodeMainPnP1stSuctionPlateVacuum.statErrorAutoCleared := FALSE;
   instCmAnodeMainPnP1stSuctionPlateVacuum.statErrorState := 16#0000;
   instCmAnodeMainPnP1stSuctionPlateVacuum.statDisablingCompleted := FALSE;
   instCmAnodeMainPnP1stSuctionPlateVacuum.statFeedbackHomePos := TRUE;
   instCmAnodeMainPnP1stSuctionPlateVacuum.statFeedbackWorkPos := FALSE;
   instCmAnodeMainPnP2ndSuctionPlateVacuum.enable := TRUE;
   instCmAnodeMainPnP2ndSuctionPlateVacuum.parentReferenceDesignator := WSTRING#'';
   instCmAnodeMainPnP2ndSuctionPlateVacuum.feedbackHomePos := TRUE;
   instCmAnodeMainPnP2ndSuctionPlateVacuum.feedbackWorkPos := FALSE;
   instCmAnodeMainPnP2ndSuctionPlateVacuum.enableManualCmds := TRUE;
   instCmAnodeMainPnP2ndSuctionPlateVacuum.interlockWorkPos := TRUE;
   instCmAnodeMainPnP2ndSuctionPlateVacuum.interlockHomePos := TRUE;
   instCmAnodeMainPnP2ndSuctionPlateVacuum.goToHomePos := FALSE;
   instCmAnodeMainPnP2ndSuctionPlateVacuum.goToWorkPos := FALSE;
   instCmAnodeMainPnP2ndSuctionPlateVacuum.statProcessValues.enable := TRUE;
   instCmAnodeMainPnP2ndSuctionPlateVacuum.statProcessValues.referenceDesignator := WSTRING#'MainPnP2Vacuum';
   instCmAnodeMainPnP2ndSuctionPlateVacuum.statProcessValues.commandHomePos := FALSE;
   instCmAnodeMainPnP2ndSuctionPlateVacuum.statProcessValues.commandWorkPos := FALSE;
   instCmAnodeMainPnP2ndSuctionPlateVacuum.statProcessValues.goToHomePos := FALSE;
   instCmAnodeMainPnP2ndSuctionPlateVacuum.statProcessValues.goToWorkPos := FALSE;
   instCmAnodeMainPnP2ndSuctionPlateVacuum.statProcessValues.inHomePos := TRUE;
   instCmAnodeMainPnP2ndSuctionPlateVacuum.statProcessValues.inWorkPos := FALSE;
   instCmAnodeMainPnP2ndSuctionPlateVacuum.statProcessValues.reset := FALSE;
   instCmAnodeMainPnP2ndSuctionPlateVacuum.statProcessValues.enableManualCmds := TRUE;
   instCmAnodeMainPnP2ndSuctionPlateVacuum.statProcessValues.error := FALSE;
   instCmAnodeMainPnP2ndSuctionPlateVacuum.statProcessValues.interlockHomePos := TRUE;
   instCmAnodeMainPnP2ndSuctionPlateVacuum.statProcessValues.interlockWorkPos := TRUE;
   instCmAnodeMainPnP2ndSuctionPlateVacuum.statProcessValues.status := 16#7003;
   instCmAnodeMainPnP2ndSuctionPlateVacuum.statProcessValues.interlockWarningWorkPos := FALSE;
   instCmAnodeMainPnP2ndSuctionPlateVacuum.statProcessValues.interlockWarningHomePos := FALSE;
   instCmAnodeMainPnP2ndSuctionPlateVacuum.statCurrentInputs.commandHomePos := FALSE;
   instCmAnodeMainPnP2ndSuctionPlateVacuum.statCurrentInputs.commandWorkPos := FALSE;
   instCmAnodeMainPnP2ndSuctionPlateVacuum.statCurrentInputs.reset := FALSE;
   instCmAnodeMainPnP2ndSuctionPlateVacuum.statPreviousInputs.commandHomePos := FALSE;
   instCmAnodeMainPnP2ndSuctionPlateVacuum.statPreviousInputs.commandWorkPos := FALSE;
   instCmAnodeMainPnP2ndSuctionPlateVacuum.statPreviousInputs.reset := FALSE;
   instCmAnodeMainPnP2ndSuctionPlateVacuum.statCurrentInterface.commandHomePos := FALSE;
   instCmAnodeMainPnP2ndSuctionPlateVacuum.statCurrentInterface.commandWorkPos := FALSE;
   instCmAnodeMainPnP2ndSuctionPlateVacuum.statCurrentInterface.reset := FALSE;
   instCmAnodeMainPnP2ndSuctionPlateVacuum.statPreviousInterface.commandHomePos := FALSE;
   instCmAnodeMainPnP2ndSuctionPlateVacuum.statPreviousInterface.commandWorkPos := FALSE;
   instCmAnodeMainPnP2ndSuctionPlateVacuum.statPreviousInterface.reset := FALSE;
   instCmAnodeMainPnP2ndSuctionPlateVacuum.statEmptyDiagnostics.status := 16#0000;
   instCmAnodeMainPnP2ndSuctionPlateVacuum.statEmptyDiagnostics.subfunctionStatus := 16#0000;
   instCmAnodeMainPnP2ndSuctionPlateVacuum.statEmptyDiagnostics.stateNumber := 0;
   instCmAnodeMainPnP2ndSuctionPlateVacuum.instTimerReachPos.PT := T#0MS;
   instCmAnodeMainPnP2ndSuctionPlateVacuum.instTimerReachPos.IN := FALSE;
   instCmAnodeMainPnP2ndSuctionPlateVacuum.instTimerLeavePos.PT := T#0MS;
   instCmAnodeMainPnP2ndSuctionPlateVacuum.instTimerLeavePos.IN := FALSE;
   instCmAnodeMainPnP2ndSuctionPlateVacuum.instTimerDiscrepancyCheck.PT := T#0MS;
   instCmAnodeMainPnP2ndSuctionPlateVacuum.instTimerDiscrepancyCheck.IN := FALSE;
   instCmAnodeMainPnP2ndSuctionPlateVacuum.statDisableAlarms := FALSE;
   instCmAnodeMainPnP2ndSuctionPlateVacuum.statDiagnostics.status := 16#7003;
   instCmAnodeMainPnP2ndSuctionPlateVacuum.statDiagnostics.subfunctionStatus := 16#0000;
   instCmAnodeMainPnP2ndSuctionPlateVacuum.statDiagnostics.stateNumber := 0;
   instCmAnodeMainPnP2ndSuctionPlateVacuum.statEnablePrevious := TRUE;
   instCmAnodeMainPnP2ndSuctionPlateVacuum.statFirstCall := FALSE;
   instCmAnodeMainPnP2ndSuctionPlateVacuum.statResetPrevious := FALSE;
   instCmAnodeMainPnP2ndSuctionPlateVacuum.statValid := TRUE;
   instCmAnodeMainPnP2ndSuctionPlateVacuum.statBusy := TRUE;
   instCmAnodeMainPnP2ndSuctionPlateVacuum.statError := FALSE;
   instCmAnodeMainPnP2ndSuctionPlateVacuum.statInterlockWorkOff := FALSE;
   instCmAnodeMainPnP2ndSuctionPlateVacuum.statInterlockHomeOff := FALSE;
   instCmAnodeMainPnP2ndSuctionPlateVacuum.statFbState := 50;
   instCmAnodeMainPnP2ndSuctionPlateVacuum.statFbStatePrevious := 50;
   instCmAnodeMainPnP2ndSuctionPlateVacuum.statErrorUserCleared := FALSE;
   instCmAnodeMainPnP2ndSuctionPlateVacuum.statErrorAutoCleared := FALSE;
   instCmAnodeMainPnP2ndSuctionPlateVacuum.statErrorState := 16#0000;
   instCmAnodeMainPnP2ndSuctionPlateVacuum.statDisablingCompleted := FALSE;
   instCmAnodeMainPnP2ndSuctionPlateVacuum.statFeedbackHomePos := TRUE;
   instCmAnodeMainPnP2ndSuctionPlateVacuum.statFeedbackWorkPos := FALSE;
   instCmAnodeAlignTableSuctionPlateVacuum.enable := TRUE;
   instCmAnodeAlignTableSuctionPlateVacuum.parentReferenceDesignator := WSTRING#'';
   instCmAnodeAlignTableSuctionPlateVacuum.feedbackHomePos := TRUE;
   instCmAnodeAlignTableSuctionPlateVacuum.feedbackWorkPos := FALSE;
   instCmAnodeAlignTableSuctionPlateVacuum.enableManualCmds := TRUE;
   instCmAnodeAlignTableSuctionPlateVacuum.interlockWorkPos := TRUE;
   instCmAnodeAlignTableSuctionPlateVacuum.interlockHomePos := TRUE;
   instCmAnodeAlignTableSuctionPlateVacuum.goToHomePos := FALSE;
   instCmAnodeAlignTableSuctionPlateVacuum.goToWorkPos := FALSE;
   instCmAnodeAlignTableSuctionPlateVacuum.statProcessValues.enable := TRUE;
   instCmAnodeAlignTableSuctionPlateVacuum.statProcessValues.referenceDesignator := WSTRING#'AlignTableVaccum';
   instCmAnodeAlignTableSuctionPlateVacuum.statProcessValues.commandHomePos := FALSE;
   instCmAnodeAlignTableSuctionPlateVacuum.statProcessValues.commandWorkPos := FALSE;
   instCmAnodeAlignTableSuctionPlateVacuum.statProcessValues.goToHomePos := FALSE;
   instCmAnodeAlignTableSuctionPlateVacuum.statProcessValues.goToWorkPos := FALSE;
   instCmAnodeAlignTableSuctionPlateVacuum.statProcessValues.inHomePos := TRUE;
   instCmAnodeAlignTableSuctionPlateVacuum.statProcessValues.inWorkPos := FALSE;
   instCmAnodeAlignTableSuctionPlateVacuum.statProcessValues.reset := FALSE;
   instCmAnodeAlignTableSuctionPlateVacuum.statProcessValues.enableManualCmds := TRUE;
   instCmAnodeAlignTableSuctionPlateVacuum.statProcessValues.error := FALSE;
   instCmAnodeAlignTableSuctionPlateVacuum.statProcessValues.interlockHomePos := TRUE;
   instCmAnodeAlignTableSuctionPlateVacuum.statProcessValues.interlockWorkPos := TRUE;
   instCmAnodeAlignTableSuctionPlateVacuum.statProcessValues.status := 16#7003;
   instCmAnodeAlignTableSuctionPlateVacuum.statProcessValues.interlockWarningWorkPos := FALSE;
   instCmAnodeAlignTableSuctionPlateVacuum.statProcessValues.interlockWarningHomePos := FALSE;
   instCmAnodeAlignTableSuctionPlateVacuum.statCurrentInputs.commandHomePos := FALSE;
   instCmAnodeAlignTableSuctionPlateVacuum.statCurrentInputs.commandWorkPos := FALSE;
   instCmAnodeAlignTableSuctionPlateVacuum.statCurrentInputs.reset := FALSE;
   instCmAnodeAlignTableSuctionPlateVacuum.statPreviousInputs.commandHomePos := FALSE;
   instCmAnodeAlignTableSuctionPlateVacuum.statPreviousInputs.commandWorkPos := FALSE;
   instCmAnodeAlignTableSuctionPlateVacuum.statPreviousInputs.reset := FALSE;
   instCmAnodeAlignTableSuctionPlateVacuum.statCurrentInterface.commandHomePos := FALSE;
   instCmAnodeAlignTableSuctionPlateVacuum.statCurrentInterface.commandWorkPos := FALSE;
   instCmAnodeAlignTableSuctionPlateVacuum.statCurrentInterface.reset := FALSE;
   instCmAnodeAlignTableSuctionPlateVacuum.statPreviousInterface.commandHomePos := FALSE;
   instCmAnodeAlignTableSuctionPlateVacuum.statPreviousInterface.commandWorkPos := FALSE;
   instCmAnodeAlignTableSuctionPlateVacuum.statPreviousInterface.reset := FALSE;
   instCmAnodeAlignTableSuctionPlateVacuum.statEmptyDiagnostics.status := 16#0000;
   instCmAnodeAlignTableSuctionPlateVacuum.statEmptyDiagnostics.subfunctionStatus := 16#0000;
   instCmAnodeAlignTableSuctionPlateVacuum.statEmptyDiagnostics.stateNumber := 0;
   instCmAnodeAlignTableSuctionPlateVacuum.instTimerReachPos.PT := T#0MS;
   instCmAnodeAlignTableSuctionPlateVacuum.instTimerReachPos.IN := FALSE;
   instCmAnodeAlignTableSuctionPlateVacuum.instTimerLeavePos.PT := T#0MS;
   instCmAnodeAlignTableSuctionPlateVacuum.instTimerLeavePos.IN := FALSE;
   instCmAnodeAlignTableSuctionPlateVacuum.instTimerDiscrepancyCheck.PT := T#0MS;
   instCmAnodeAlignTableSuctionPlateVacuum.instTimerDiscrepancyCheck.IN := FALSE;
   instCmAnodeAlignTableSuctionPlateVacuum.statDisableAlarms := FALSE;
   instCmAnodeAlignTableSuctionPlateVacuum.statDiagnostics.status := 16#7003;
   instCmAnodeAlignTableSuctionPlateVacuum.statDiagnostics.subfunctionStatus := 16#0000;
   instCmAnodeAlignTableSuctionPlateVacuum.statDiagnostics.stateNumber := 0;
   instCmAnodeAlignTableSuctionPlateVacuum.statEnablePrevious := TRUE;
   instCmAnodeAlignTableSuctionPlateVacuum.statFirstCall := FALSE;
   instCmAnodeAlignTableSuctionPlateVacuum.statResetPrevious := FALSE;
   instCmAnodeAlignTableSuctionPlateVacuum.statValid := TRUE;
   instCmAnodeAlignTableSuctionPlateVacuum.statBusy := TRUE;
   instCmAnodeAlignTableSuctionPlateVacuum.statError := FALSE;
   instCmAnodeAlignTableSuctionPlateVacuum.statInterlockWorkOff := FALSE;
   instCmAnodeAlignTableSuctionPlateVacuum.statInterlockHomeOff := FALSE;
   instCmAnodeAlignTableSuctionPlateVacuum.statFbState := 50;
   instCmAnodeAlignTableSuctionPlateVacuum.statFbStatePrevious := 50;
   instCmAnodeAlignTableSuctionPlateVacuum.statErrorUserCleared := FALSE;
   instCmAnodeAlignTableSuctionPlateVacuum.statErrorAutoCleared := FALSE;
   instCmAnodeAlignTableSuctionPlateVacuum.statErrorState := 16#0000;
   instCmAnodeAlignTableSuctionPlateVacuum.statDisablingCompleted := FALSE;
   instCmAnodeAlignTableSuctionPlateVacuum.statFeedbackHomePos := TRUE;
   instCmAnodeAlignTableSuctionPlateVacuum.statFeedbackWorkPos := FALSE;
   instCmAnodeGlassCleaning.enable := TRUE;
   instCmAnodeGlassCleaning.parentReferenceDesignator := WSTRING#'';
   instCmAnodeGlassCleaning.feedbackHomePos := FALSE;
   instCmAnodeGlassCleaning.feedbackWorkPos := FALSE;
   instCmAnodeGlassCleaning.enableManualCmds := TRUE;
   instCmAnodeGlassCleaning.interlockWorkPos := TRUE;
   instCmAnodeGlassCleaning.interlockHomePos := TRUE;
   instCmAnodeGlassCleaning.goToHomePos := FALSE;
   instCmAnodeGlassCleaning.goToWorkPos := FALSE;
   instCmAnodeGlassCleaning.statProcessValues.enable := TRUE;
   instCmAnodeGlassCleaning.statProcessValues.referenceDesignator := WSTRING#'GlassCleaning';
   instCmAnodeGlassCleaning.statProcessValues.commandHomePos := FALSE;
   instCmAnodeGlassCleaning.statProcessValues.commandWorkPos := FALSE;
   instCmAnodeGlassCleaning.statProcessValues.goToHomePos := FALSE;
   instCmAnodeGlassCleaning.statProcessValues.goToWorkPos := FALSE;
   instCmAnodeGlassCleaning.statProcessValues.inHomePos := FALSE;
   instCmAnodeGlassCleaning.statProcessValues.inWorkPos := FALSE;
   instCmAnodeGlassCleaning.statProcessValues.reset := FALSE;
   instCmAnodeGlassCleaning.statProcessValues.enableManualCmds := TRUE;
   instCmAnodeGlassCleaning.statProcessValues.error := FALSE;
   instCmAnodeGlassCleaning.statProcessValues.interlockHomePos := TRUE;
   instCmAnodeGlassCleaning.statProcessValues.interlockWorkPos := TRUE;
   instCmAnodeGlassCleaning.statProcessValues.status := 16#7003;
   instCmAnodeGlassCleaning.statProcessValues.interlockWarningWorkPos := FALSE;
   instCmAnodeGlassCleaning.statProcessValues.interlockWarningHomePos := FALSE;
   instCmAnodeGlassCleaning.statCurrentInputs.commandHomePos := FALSE;
   instCmAnodeGlassCleaning.statCurrentInputs.commandWorkPos := FALSE;
   instCmAnodeGlassCleaning.statCurrentInputs.reset := FALSE;
   instCmAnodeGlassCleaning.statPreviousInputs.commandHomePos := FALSE;
   instCmAnodeGlassCleaning.statPreviousInputs.commandWorkPos := FALSE;
   instCmAnodeGlassCleaning.statPreviousInputs.reset := FALSE;
   instCmAnodeGlassCleaning.statCurrentInterface.commandHomePos := FALSE;
   instCmAnodeGlassCleaning.statCurrentInterface.commandWorkPos := FALSE;
   instCmAnodeGlassCleaning.statCurrentInterface.reset := FALSE;
   instCmAnodeGlassCleaning.statPreviousInterface.commandHomePos := FALSE;
   instCmAnodeGlassCleaning.statPreviousInterface.commandWorkPos := FALSE;
   instCmAnodeGlassCleaning.statPreviousInterface.reset := FALSE;
   instCmAnodeGlassCleaning.statEmptyDiagnostics.status := 16#0000;
   instCmAnodeGlassCleaning.statEmptyDiagnostics.subfunctionStatus := 16#0000;
   instCmAnodeGlassCleaning.statEmptyDiagnostics.stateNumber := 0;
   instCmAnodeGlassCleaning.instTimerReachPos.PT := T#0MS;
   instCmAnodeGlassCleaning.instTimerReachPos.IN := FALSE;
   instCmAnodeGlassCleaning.instTimerLeavePos.PT := T#0MS;
   instCmAnodeGlassCleaning.instTimerLeavePos.IN := FALSE;
   instCmAnodeGlassCleaning.instTimerDiscrepancyCheck.PT := T#0MS;
   instCmAnodeGlassCleaning.instTimerDiscrepancyCheck.IN := FALSE;
   instCmAnodeGlassCleaning.statDisableAlarms := FALSE;
   instCmAnodeGlassCleaning.statDiagnostics.status := 16#7003;
   instCmAnodeGlassCleaning.statDiagnostics.subfunctionStatus := 16#0000;
   instCmAnodeGlassCleaning.statDiagnostics.stateNumber := 0;
   instCmAnodeGlassCleaning.statEnablePrevious := TRUE;
   instCmAnodeGlassCleaning.statFirstCall := FALSE;
   instCmAnodeGlassCleaning.statResetPrevious := FALSE;
   instCmAnodeGlassCleaning.statValid := TRUE;
   instCmAnodeGlassCleaning.statBusy := TRUE;
   instCmAnodeGlassCleaning.statError := FALSE;
   instCmAnodeGlassCleaning.statInterlockWorkOff := FALSE;
   instCmAnodeGlassCleaning.statInterlockHomeOff := FALSE;
   instCmAnodeGlassCleaning.statFbState := 50;
   instCmAnodeGlassCleaning.statFbStatePrevious := 50;
   instCmAnodeGlassCleaning.statErrorUserCleared := FALSE;
   instCmAnodeGlassCleaning.statErrorAutoCleared := FALSE;
   instCmAnodeGlassCleaning.statErrorState := 16#0000;
   instCmAnodeGlassCleaning.statDisablingCompleted := FALSE;
   instCmAnodeGlassCleaning.statFeedbackHomePos := FALSE;
   instCmAnodeGlassCleaning.statFeedbackWorkPos := FALSE;
   instCmAnodeNgPnpUpDown.enable := TRUE;
   instCmAnodeNgPnpUpDown.parentReferenceDesignator := WSTRING#'';
   instCmAnodeNgPnpUpDown.feedbackHomePos := TRUE;
   instCmAnodeNgPnpUpDown.feedbackWorkPos := FALSE;
   instCmAnodeNgPnpUpDown.enableManualCmds := TRUE;
   instCmAnodeNgPnpUpDown.interlockWorkPos := FALSE;
   instCmAnodeNgPnpUpDown.interlockHomePos := TRUE;
   instCmAnodeNgPnpUpDown.goToHomePos := FALSE;
   instCmAnodeNgPnpUpDown.goToWorkPos := FALSE;
   instCmAnodeNgPnpUpDown.statProcessValues.enable := TRUE;
   instCmAnodeNgPnpUpDown.statProcessValues.referenceDesignator := WSTRING#'NgPnpUpDown';
   instCmAnodeNgPnpUpDown.statProcessValues.commandHomePos := FALSE;
   instCmAnodeNgPnpUpDown.statProcessValues.commandWorkPos := FALSE;
   instCmAnodeNgPnpUpDown.statProcessValues.goToHomePos := FALSE;
   instCmAnodeNgPnpUpDown.statProcessValues.goToWorkPos := FALSE;
   instCmAnodeNgPnpUpDown.statProcessValues.inHomePos := FALSE;
   instCmAnodeNgPnpUpDown.statProcessValues.inWorkPos := FALSE;
   instCmAnodeNgPnpUpDown.statProcessValues.reset := FALSE;
   instCmAnodeNgPnpUpDown.statProcessValues.enableManualCmds := TRUE;
   instCmAnodeNgPnpUpDown.statProcessValues.error := FALSE;
   instCmAnodeNgPnpUpDown.statProcessValues.interlockHomePos := TRUE;
   instCmAnodeNgPnpUpDown.statProcessValues.interlockWorkPos := FALSE;
   instCmAnodeNgPnpUpDown.statProcessValues.status := 16#7101;
   instCmAnodeNgPnpUpDown.statProcessValues.interlockWarningWorkPos := FALSE;
   instCmAnodeNgPnpUpDown.statProcessValues.interlockWarningHomePos := FALSE;
   instCmAnodeNgPnpUpDown.statCurrentInputs.commandHomePos := FALSE;
   instCmAnodeNgPnpUpDown.statCurrentInputs.commandWorkPos := FALSE;
   instCmAnodeNgPnpUpDown.statCurrentInputs.reset := FALSE;
   instCmAnodeNgPnpUpDown.statPreviousInputs.commandHomePos := FALSE;
   instCmAnodeNgPnpUpDown.statPreviousInputs.commandWorkPos := FALSE;
   instCmAnodeNgPnpUpDown.statPreviousInputs.reset := FALSE;
   instCmAnodeNgPnpUpDown.statCurrentInterface.commandHomePos := FALSE;
   instCmAnodeNgPnpUpDown.statCurrentInterface.commandWorkPos := FALSE;
   instCmAnodeNgPnpUpDown.statCurrentInterface.reset := FALSE;
   instCmAnodeNgPnpUpDown.statPreviousInterface.commandHomePos := FALSE;
   instCmAnodeNgPnpUpDown.statPreviousInterface.commandWorkPos := FALSE;
   instCmAnodeNgPnpUpDown.statPreviousInterface.reset := FALSE;
   instCmAnodeNgPnpUpDown.statEmptyDiagnostics.status := 16#0000;
   instCmAnodeNgPnpUpDown.statEmptyDiagnostics.subfunctionStatus := 16#0000;
   instCmAnodeNgPnpUpDown.statEmptyDiagnostics.stateNumber := 0;
   instCmAnodeNgPnpUpDown.instTimerReachPos.PT := T#0MS;
   instCmAnodeNgPnpUpDown.instTimerReachPos.IN := FALSE;
   instCmAnodeNgPnpUpDown.instTimerLeavePos.PT := T#0MS;
   instCmAnodeNgPnpUpDown.instTimerLeavePos.IN := FALSE;
   instCmAnodeNgPnpUpDown.instTimerDiscrepancyCheck.PT := T#0MS;
   instCmAnodeNgPnpUpDown.instTimerDiscrepancyCheck.IN := FALSE;
   instCmAnodeNgPnpUpDown.statDisableAlarms := FALSE;
   instCmAnodeNgPnpUpDown.statDiagnostics.status := 16#7003;
   instCmAnodeNgPnpUpDown.statDiagnostics.subfunctionStatus := 16#0000;
   instCmAnodeNgPnpUpDown.statDiagnostics.stateNumber := 0;
   instCmAnodeNgPnpUpDown.statEnablePrevious := TRUE;
   instCmAnodeNgPnpUpDown.statFirstCall := FALSE;
   instCmAnodeNgPnpUpDown.statResetPrevious := FALSE;
   instCmAnodeNgPnpUpDown.statValid := TRUE;
   instCmAnodeNgPnpUpDown.statBusy := TRUE;
   instCmAnodeNgPnpUpDown.statError := FALSE;
   instCmAnodeNgPnpUpDown.statInterlockWorkOff := FALSE;
   instCmAnodeNgPnpUpDown.statInterlockHomeOff := FALSE;
   instCmAnodeNgPnpUpDown.statFbState := 50;
   instCmAnodeNgPnpUpDown.statFbStatePrevious := 50;
   instCmAnodeNgPnpUpDown.statErrorUserCleared := FALSE;
   instCmAnodeNgPnpUpDown.statErrorAutoCleared := FALSE;
   instCmAnodeNgPnpUpDown.statErrorState := 16#0000;
   instCmAnodeNgPnpUpDown.statDisablingCompleted := FALSE;
   instCmAnodeNgPnpUpDown.statFeedbackHomePos := TRUE;
   instCmAnodeNgPnpUpDown.statFeedbackWorkPos := FALSE;
   instCmAnodeNgPnp1stFwdBwd.enable := TRUE;
   instCmAnodeNgPnp1stFwdBwd.parentReferenceDesignator := WSTRING#'';
   instCmAnodeNgPnp1stFwdBwd.feedbackHomePos := FALSE;
   instCmAnodeNgPnp1stFwdBwd.feedbackWorkPos := FALSE;
   instCmAnodeNgPnp1stFwdBwd.enableManualCmds := TRUE;
   instCmAnodeNgPnp1stFwdBwd.interlockWorkPos := FALSE;
   instCmAnodeNgPnp1stFwdBwd.interlockHomePos := TRUE;
   instCmAnodeNgPnp1stFwdBwd.goToHomePos := FALSE;
   instCmAnodeNgPnp1stFwdBwd.goToWorkPos := FALSE;
   instCmAnodeNgPnp1stFwdBwd.statProcessValues.enable := TRUE;
   instCmAnodeNgPnp1stFwdBwd.statProcessValues.referenceDesignator := WSTRING#'NgPnp1stFwdBwd';
   instCmAnodeNgPnp1stFwdBwd.statProcessValues.commandHomePos := FALSE;
   instCmAnodeNgPnp1stFwdBwd.statProcessValues.commandWorkPos := FALSE;
   instCmAnodeNgPnp1stFwdBwd.statProcessValues.goToHomePos := FALSE;
   instCmAnodeNgPnp1stFwdBwd.statProcessValues.goToWorkPos := FALSE;
   instCmAnodeNgPnp1stFwdBwd.statProcessValues.inHomePos := FALSE;
   instCmAnodeNgPnp1stFwdBwd.statProcessValues.inWorkPos := FALSE;
   instCmAnodeNgPnp1stFwdBwd.statProcessValues.reset := FALSE;
   instCmAnodeNgPnp1stFwdBwd.statProcessValues.enableManualCmds := TRUE;
   instCmAnodeNgPnp1stFwdBwd.statProcessValues.error := FALSE;
   instCmAnodeNgPnp1stFwdBwd.statProcessValues.interlockHomePos := TRUE;
   instCmAnodeNgPnp1stFwdBwd.statProcessValues.interlockWorkPos := FALSE;
   instCmAnodeNgPnp1stFwdBwd.statProcessValues.status := 16#7101;
   instCmAnodeNgPnp1stFwdBwd.statProcessValues.interlockWarningWorkPos := FALSE;
   instCmAnodeNgPnp1stFwdBwd.statProcessValues.interlockWarningHomePos := FALSE;
   instCmAnodeNgPnp1stFwdBwd.statCurrentInputs.commandHomePos := FALSE;
   instCmAnodeNgPnp1stFwdBwd.statCurrentInputs.commandWorkPos := FALSE;
   instCmAnodeNgPnp1stFwdBwd.statCurrentInputs.reset := FALSE;
   instCmAnodeNgPnp1stFwdBwd.statPreviousInputs.commandHomePos := FALSE;
   instCmAnodeNgPnp1stFwdBwd.statPreviousInputs.commandWorkPos := FALSE;
   instCmAnodeNgPnp1stFwdBwd.statPreviousInputs.reset := FALSE;
   instCmAnodeNgPnp1stFwdBwd.statCurrentInterface.commandHomePos := FALSE;
   instCmAnodeNgPnp1stFwdBwd.statCurrentInterface.commandWorkPos := FALSE;
   instCmAnodeNgPnp1stFwdBwd.statCurrentInterface.reset := FALSE;
   instCmAnodeNgPnp1stFwdBwd.statPreviousInterface.commandHomePos := FALSE;
   instCmAnodeNgPnp1stFwdBwd.statPreviousInterface.commandWorkPos := FALSE;
   instCmAnodeNgPnp1stFwdBwd.statPreviousInterface.reset := FALSE;
   instCmAnodeNgPnp1stFwdBwd.statEmptyDiagnostics.status := 16#0000;
   instCmAnodeNgPnp1stFwdBwd.statEmptyDiagnostics.subfunctionStatus := 16#0000;
   instCmAnodeNgPnp1stFwdBwd.statEmptyDiagnostics.stateNumber := 0;
   instCmAnodeNgPnp1stFwdBwd.instTimerReachPos.PT := T#0MS;
   instCmAnodeNgPnp1stFwdBwd.instTimerReachPos.IN := FALSE;
   instCmAnodeNgPnp1stFwdBwd.instTimerLeavePos.PT := T#0MS;
   instCmAnodeNgPnp1stFwdBwd.instTimerLeavePos.IN := FALSE;
   instCmAnodeNgPnp1stFwdBwd.instTimerDiscrepancyCheck.PT := T#0MS;
   instCmAnodeNgPnp1stFwdBwd.instTimerDiscrepancyCheck.IN := FALSE;
   instCmAnodeNgPnp1stFwdBwd.statDisableAlarms := FALSE;
   instCmAnodeNgPnp1stFwdBwd.statDiagnostics.status := 16#7003;
   instCmAnodeNgPnp1stFwdBwd.statDiagnostics.subfunctionStatus := 16#0000;
   instCmAnodeNgPnp1stFwdBwd.statDiagnostics.stateNumber := 0;
   instCmAnodeNgPnp1stFwdBwd.statEnablePrevious := TRUE;
   instCmAnodeNgPnp1stFwdBwd.statFirstCall := FALSE;
   instCmAnodeNgPnp1stFwdBwd.statResetPrevious := FALSE;
   instCmAnodeNgPnp1stFwdBwd.statValid := TRUE;
   instCmAnodeNgPnp1stFwdBwd.statBusy := TRUE;
   instCmAnodeNgPnp1stFwdBwd.statError := FALSE;
   instCmAnodeNgPnp1stFwdBwd.statInterlockWorkOff := FALSE;
   instCmAnodeNgPnp1stFwdBwd.statInterlockHomeOff := FALSE;
   instCmAnodeNgPnp1stFwdBwd.statFbState := 50;
   instCmAnodeNgPnp1stFwdBwd.statFbStatePrevious := 50;
   instCmAnodeNgPnp1stFwdBwd.statErrorUserCleared := FALSE;
   instCmAnodeNgPnp1stFwdBwd.statErrorAutoCleared := FALSE;
   instCmAnodeNgPnp1stFwdBwd.statErrorState := 16#0000;
   instCmAnodeNgPnp1stFwdBwd.statDisablingCompleted := FALSE;
   instCmAnodeNgPnp1stFwdBwd.statFeedbackHomePos := FALSE;
   instCmAnodeNgPnp1stFwdBwd.statFeedbackWorkPos := FALSE;
   instCmAnodeNgPnp2ndFwdBwd.enable := TRUE;
   instCmAnodeNgPnp2ndFwdBwd.parentReferenceDesignator := WSTRING#'';
   instCmAnodeNgPnp2ndFwdBwd.feedbackHomePos := FALSE;
   instCmAnodeNgPnp2ndFwdBwd.feedbackWorkPos := FALSE;
   instCmAnodeNgPnp2ndFwdBwd.enableManualCmds := TRUE;
   instCmAnodeNgPnp2ndFwdBwd.interlockWorkPos := FALSE;
   instCmAnodeNgPnp2ndFwdBwd.interlockHomePos := FALSE;
   instCmAnodeNgPnp2ndFwdBwd.goToHomePos := FALSE;
   instCmAnodeNgPnp2ndFwdBwd.goToWorkPos := FALSE;
   instCmAnodeNgPnp2ndFwdBwd.statProcessValues.enable := TRUE;
   instCmAnodeNgPnp2ndFwdBwd.statProcessValues.referenceDesignator := WSTRING#'NgPnp2ndFwdBwd';
   instCmAnodeNgPnp2ndFwdBwd.statProcessValues.commandHomePos := FALSE;
   instCmAnodeNgPnp2ndFwdBwd.statProcessValues.commandWorkPos := FALSE;
   instCmAnodeNgPnp2ndFwdBwd.statProcessValues.goToHomePos := FALSE;
   instCmAnodeNgPnp2ndFwdBwd.statProcessValues.goToWorkPos := FALSE;
   instCmAnodeNgPnp2ndFwdBwd.statProcessValues.inHomePos := FALSE;
   instCmAnodeNgPnp2ndFwdBwd.statProcessValues.inWorkPos := FALSE;
   instCmAnodeNgPnp2ndFwdBwd.statProcessValues.reset := FALSE;
   instCmAnodeNgPnp2ndFwdBwd.statProcessValues.enableManualCmds := TRUE;
   instCmAnodeNgPnp2ndFwdBwd.statProcessValues.error := FALSE;
   instCmAnodeNgPnp2ndFwdBwd.statProcessValues.interlockHomePos := FALSE;
   instCmAnodeNgPnp2ndFwdBwd.statProcessValues.interlockWorkPos := FALSE;
   instCmAnodeNgPnp2ndFwdBwd.statProcessValues.status := 16#7100;
   instCmAnodeNgPnp2ndFwdBwd.statProcessValues.interlockWarningWorkPos := FALSE;
   instCmAnodeNgPnp2ndFwdBwd.statProcessValues.interlockWarningHomePos := FALSE;
   instCmAnodeNgPnp2ndFwdBwd.statCurrentInputs.commandHomePos := FALSE;
   instCmAnodeNgPnp2ndFwdBwd.statCurrentInputs.commandWorkPos := FALSE;
   instCmAnodeNgPnp2ndFwdBwd.statCurrentInputs.reset := FALSE;
   instCmAnodeNgPnp2ndFwdBwd.statPreviousInputs.commandHomePos := FALSE;
   instCmAnodeNgPnp2ndFwdBwd.statPreviousInputs.commandWorkPos := FALSE;
   instCmAnodeNgPnp2ndFwdBwd.statPreviousInputs.reset := FALSE;
   instCmAnodeNgPnp2ndFwdBwd.statCurrentInterface.commandHomePos := FALSE;
   instCmAnodeNgPnp2ndFwdBwd.statCurrentInterface.commandWorkPos := FALSE;
   instCmAnodeNgPnp2ndFwdBwd.statCurrentInterface.reset := FALSE;
   instCmAnodeNgPnp2ndFwdBwd.statPreviousInterface.commandHomePos := FALSE;
   instCmAnodeNgPnp2ndFwdBwd.statPreviousInterface.commandWorkPos := FALSE;
   instCmAnodeNgPnp2ndFwdBwd.statPreviousInterface.reset := FALSE;
   instCmAnodeNgPnp2ndFwdBwd.statEmptyDiagnostics.status := 16#0000;
   instCmAnodeNgPnp2ndFwdBwd.statEmptyDiagnostics.subfunctionStatus := 16#0000;
   instCmAnodeNgPnp2ndFwdBwd.statEmptyDiagnostics.stateNumber := 0;
   instCmAnodeNgPnp2ndFwdBwd.instTimerReachPos.PT := T#0MS;
   instCmAnodeNgPnp2ndFwdBwd.instTimerReachPos.IN := FALSE;
   instCmAnodeNgPnp2ndFwdBwd.instTimerLeavePos.PT := T#0MS;
   instCmAnodeNgPnp2ndFwdBwd.instTimerLeavePos.IN := FALSE;
   instCmAnodeNgPnp2ndFwdBwd.instTimerDiscrepancyCheck.PT := T#0MS;
   instCmAnodeNgPnp2ndFwdBwd.instTimerDiscrepancyCheck.IN := FALSE;
   instCmAnodeNgPnp2ndFwdBwd.statDisableAlarms := FALSE;
   instCmAnodeNgPnp2ndFwdBwd.statDiagnostics.status := 16#7003;
   instCmAnodeNgPnp2ndFwdBwd.statDiagnostics.subfunctionStatus := 16#0000;
   instCmAnodeNgPnp2ndFwdBwd.statDiagnostics.stateNumber := 0;
   instCmAnodeNgPnp2ndFwdBwd.statEnablePrevious := TRUE;
   instCmAnodeNgPnp2ndFwdBwd.statFirstCall := FALSE;
   instCmAnodeNgPnp2ndFwdBwd.statResetPrevious := FALSE;
   instCmAnodeNgPnp2ndFwdBwd.statValid := TRUE;
   instCmAnodeNgPnp2ndFwdBwd.statBusy := TRUE;
   instCmAnodeNgPnp2ndFwdBwd.statError := FALSE;
   instCmAnodeNgPnp2ndFwdBwd.statInterlockWorkOff := FALSE;
   instCmAnodeNgPnp2ndFwdBwd.statInterlockHomeOff := FALSE;
   instCmAnodeNgPnp2ndFwdBwd.statFbState := 50;
   instCmAnodeNgPnp2ndFwdBwd.statFbStatePrevious := 50;
   instCmAnodeNgPnp2ndFwdBwd.statErrorUserCleared := FALSE;
   instCmAnodeNgPnp2ndFwdBwd.statErrorAutoCleared := FALSE;
   instCmAnodeNgPnp2ndFwdBwd.statErrorState := 16#0000;
   instCmAnodeNgPnp2ndFwdBwd.statDisablingCompleted := FALSE;
   instCmAnodeNgPnp2ndFwdBwd.statFeedbackHomePos := FALSE;
   instCmAnodeNgPnp2ndFwdBwd.statFeedbackWorkPos := FALSE;
   instCmAnodeMaintenanceMovingFixFwdBwd.enable := TRUE;
   instCmAnodeMaintenanceMovingFixFwdBwd.parentReferenceDesignator := WSTRING#'';
   instCmAnodeMaintenanceMovingFixFwdBwd.feedbackHomePos := TRUE;
   instCmAnodeMaintenanceMovingFixFwdBwd.feedbackWorkPos := FALSE;
   instCmAnodeMaintenanceMovingFixFwdBwd.enableManualCmds := TRUE;
   instCmAnodeMaintenanceMovingFixFwdBwd.interlockWorkPos := TRUE;
   instCmAnodeMaintenanceMovingFixFwdBwd.interlockHomePos := TRUE;
   instCmAnodeMaintenanceMovingFixFwdBwd.goToHomePos := FALSE;
   instCmAnodeMaintenanceMovingFixFwdBwd.goToWorkPos := FALSE;
   instCmAnodeMaintenanceMovingFixFwdBwd.statProcessValues.enable := TRUE;
   instCmAnodeMaintenanceMovingFixFwdBwd.statProcessValues.referenceDesignator := WSTRING#'MaintenanceFix';
   instCmAnodeMaintenanceMovingFixFwdBwd.statProcessValues.commandHomePos := FALSE;
   instCmAnodeMaintenanceMovingFixFwdBwd.statProcessValues.commandWorkPos := FALSE;
   instCmAnodeMaintenanceMovingFixFwdBwd.statProcessValues.goToHomePos := FALSE;
   instCmAnodeMaintenanceMovingFixFwdBwd.statProcessValues.goToWorkPos := FALSE;
   instCmAnodeMaintenanceMovingFixFwdBwd.statProcessValues.inHomePos := FALSE;
   instCmAnodeMaintenanceMovingFixFwdBwd.statProcessValues.inWorkPos := FALSE;
   instCmAnodeMaintenanceMovingFixFwdBwd.statProcessValues.reset := FALSE;
   instCmAnodeMaintenanceMovingFixFwdBwd.statProcessValues.enableManualCmds := TRUE;
   instCmAnodeMaintenanceMovingFixFwdBwd.statProcessValues.error := FALSE;
   instCmAnodeMaintenanceMovingFixFwdBwd.statProcessValues.interlockHomePos := TRUE;
   instCmAnodeMaintenanceMovingFixFwdBwd.statProcessValues.interlockWorkPos := TRUE;
   instCmAnodeMaintenanceMovingFixFwdBwd.statProcessValues.status := 16#7003;
   instCmAnodeMaintenanceMovingFixFwdBwd.statProcessValues.interlockWarningWorkPos := FALSE;
   instCmAnodeMaintenanceMovingFixFwdBwd.statProcessValues.interlockWarningHomePos := FALSE;
   instCmAnodeMaintenanceMovingFixFwdBwd.statCurrentInputs.commandHomePos := FALSE;
   instCmAnodeMaintenanceMovingFixFwdBwd.statCurrentInputs.commandWorkPos := FALSE;
   instCmAnodeMaintenanceMovingFixFwdBwd.statCurrentInputs.reset := FALSE;
   instCmAnodeMaintenanceMovingFixFwdBwd.statPreviousInputs.commandHomePos := FALSE;
   instCmAnodeMaintenanceMovingFixFwdBwd.statPreviousInputs.commandWorkPos := FALSE;
   instCmAnodeMaintenanceMovingFixFwdBwd.statPreviousInputs.reset := FALSE;
   instCmAnodeMaintenanceMovingFixFwdBwd.statCurrentInterface.commandHomePos := FALSE;
   instCmAnodeMaintenanceMovingFixFwdBwd.statCurrentInterface.commandWorkPos := FALSE;
   instCmAnodeMaintenanceMovingFixFwdBwd.statCurrentInterface.reset := FALSE;
   instCmAnodeMaintenanceMovingFixFwdBwd.statPreviousInterface.commandHomePos := FALSE;
   instCmAnodeMaintenanceMovingFixFwdBwd.statPreviousInterface.commandWorkPos := FALSE;
   instCmAnodeMaintenanceMovingFixFwdBwd.statPreviousInterface.reset := FALSE;
   instCmAnodeMaintenanceMovingFixFwdBwd.statEmptyDiagnostics.status := 16#0000;
   instCmAnodeMaintenanceMovingFixFwdBwd.statEmptyDiagnostics.subfunctionStatus := 16#0000;
   instCmAnodeMaintenanceMovingFixFwdBwd.statEmptyDiagnostics.stateNumber := 0;
   instCmAnodeMaintenanceMovingFixFwdBwd.instTimerReachPos.PT := T#0MS;
   instCmAnodeMaintenanceMovingFixFwdBwd.instTimerReachPos.IN := FALSE;
   instCmAnodeMaintenanceMovingFixFwdBwd.instTimerLeavePos.PT := T#0MS;
   instCmAnodeMaintenanceMovingFixFwdBwd.instTimerLeavePos.IN := FALSE;
   instCmAnodeMaintenanceMovingFixFwdBwd.instTimerDiscrepancyCheck.PT := T#0MS;
   instCmAnodeMaintenanceMovingFixFwdBwd.instTimerDiscrepancyCheck.IN := FALSE;
   instCmAnodeMaintenanceMovingFixFwdBwd.statDisableAlarms := FALSE;
   instCmAnodeMaintenanceMovingFixFwdBwd.statDiagnostics.status := 16#7003;
   instCmAnodeMaintenanceMovingFixFwdBwd.statDiagnostics.subfunctionStatus := 16#0000;
   instCmAnodeMaintenanceMovingFixFwdBwd.statDiagnostics.stateNumber := 0;
   instCmAnodeMaintenanceMovingFixFwdBwd.statEnablePrevious := TRUE;
   instCmAnodeMaintenanceMovingFixFwdBwd.statFirstCall := FALSE;
   instCmAnodeMaintenanceMovingFixFwdBwd.statResetPrevious := FALSE;
   instCmAnodeMaintenanceMovingFixFwdBwd.statValid := TRUE;
   instCmAnodeMaintenanceMovingFixFwdBwd.statBusy := TRUE;
   instCmAnodeMaintenanceMovingFixFwdBwd.statError := FALSE;
   instCmAnodeMaintenanceMovingFixFwdBwd.statInterlockWorkOff := FALSE;
   instCmAnodeMaintenanceMovingFixFwdBwd.statInterlockHomeOff := FALSE;
   instCmAnodeMaintenanceMovingFixFwdBwd.statFbState := 50;
   instCmAnodeMaintenanceMovingFixFwdBwd.statFbStatePrevious := 50;
   instCmAnodeMaintenanceMovingFixFwdBwd.statErrorUserCleared := FALSE;
   instCmAnodeMaintenanceMovingFixFwdBwd.statErrorAutoCleared := FALSE;
   instCmAnodeMaintenanceMovingFixFwdBwd.statErrorState := 16#0000;
   instCmAnodeMaintenanceMovingFixFwdBwd.statDisablingCompleted := FALSE;
   instCmAnodeMaintenanceMovingFixFwdBwd.statFeedbackHomePos := TRUE;
   instCmAnodeMaintenanceMovingFixFwdBwd.statFeedbackWorkPos := FALSE;
   instCmAnodeNgBoxLiftUpDown.enable := TRUE;
   instCmAnodeNgBoxLiftUpDown.parentReferenceDesignator := WSTRING#'';
   instCmAnodeNgBoxLiftUpDown.feedbackHomePos := TRUE;
   instCmAnodeNgBoxLiftUpDown.feedbackWorkPos := FALSE;
   instCmAnodeNgBoxLiftUpDown.enableManualCmds := TRUE;
   instCmAnodeNgBoxLiftUpDown.interlockWorkPos := FALSE;
   instCmAnodeNgBoxLiftUpDown.interlockHomePos := TRUE;
   instCmAnodeNgBoxLiftUpDown.goToHomePos := FALSE;
   instCmAnodeNgBoxLiftUpDown.goToWorkPos := FALSE;
   instCmAnodeNgBoxLiftUpDown.statProcessValues.enable := TRUE;
   instCmAnodeNgBoxLiftUpDown.statProcessValues.referenceDesignator := WSTRING#'NgBoxLiftUpDown';
   instCmAnodeNgBoxLiftUpDown.statProcessValues.commandHomePos := FALSE;
   instCmAnodeNgBoxLiftUpDown.statProcessValues.commandWorkPos := FALSE;
   instCmAnodeNgBoxLiftUpDown.statProcessValues.goToHomePos := FALSE;
   instCmAnodeNgBoxLiftUpDown.statProcessValues.goToWorkPos := FALSE;
   instCmAnodeNgBoxLiftUpDown.statProcessValues.inHomePos := FALSE;
   instCmAnodeNgBoxLiftUpDown.statProcessValues.inWorkPos := FALSE;
   instCmAnodeNgBoxLiftUpDown.statProcessValues.reset := FALSE;
   instCmAnodeNgBoxLiftUpDown.statProcessValues.enableManualCmds := TRUE;
   instCmAnodeNgBoxLiftUpDown.statProcessValues.error := FALSE;
   instCmAnodeNgBoxLiftUpDown.statProcessValues.interlockHomePos := TRUE;
   instCmAnodeNgBoxLiftUpDown.statProcessValues.interlockWorkPos := FALSE;
   instCmAnodeNgBoxLiftUpDown.statProcessValues.status := 16#7101;
   instCmAnodeNgBoxLiftUpDown.statProcessValues.interlockWarningWorkPos := FALSE;
   instCmAnodeNgBoxLiftUpDown.statProcessValues.interlockWarningHomePos := FALSE;
   instCmAnodeNgBoxLiftUpDown.statCurrentInputs.commandHomePos := FALSE;
   instCmAnodeNgBoxLiftUpDown.statCurrentInputs.commandWorkPos := FALSE;
   instCmAnodeNgBoxLiftUpDown.statCurrentInputs.reset := FALSE;
   instCmAnodeNgBoxLiftUpDown.statPreviousInputs.commandHomePos := FALSE;
   instCmAnodeNgBoxLiftUpDown.statPreviousInputs.commandWorkPos := FALSE;
   instCmAnodeNgBoxLiftUpDown.statPreviousInputs.reset := FALSE;
   instCmAnodeNgBoxLiftUpDown.statCurrentInterface.commandHomePos := FALSE;
   instCmAnodeNgBoxLiftUpDown.statCurrentInterface.commandWorkPos := FALSE;
   instCmAnodeNgBoxLiftUpDown.statCurrentInterface.reset := FALSE;
   instCmAnodeNgBoxLiftUpDown.statPreviousInterface.commandHomePos := FALSE;
   instCmAnodeNgBoxLiftUpDown.statPreviousInterface.commandWorkPos := FALSE;
   instCmAnodeNgBoxLiftUpDown.statPreviousInterface.reset := FALSE;
   instCmAnodeNgBoxLiftUpDown.statEmptyDiagnostics.status := 16#0000;
   instCmAnodeNgBoxLiftUpDown.statEmptyDiagnostics.subfunctionStatus := 16#0000;
   instCmAnodeNgBoxLiftUpDown.statEmptyDiagnostics.stateNumber := 0;
   instCmAnodeNgBoxLiftUpDown.instTimerReachPos.PT := T#0MS;
   instCmAnodeNgBoxLiftUpDown.instTimerReachPos.IN := FALSE;
   instCmAnodeNgBoxLiftUpDown.instTimerLeavePos.PT := T#0MS;
   instCmAnodeNgBoxLiftUpDown.instTimerLeavePos.IN := FALSE;
   instCmAnodeNgBoxLiftUpDown.instTimerDiscrepancyCheck.PT := T#0MS;
   instCmAnodeNgBoxLiftUpDown.instTimerDiscrepancyCheck.IN := FALSE;
   instCmAnodeNgBoxLiftUpDown.statDisableAlarms := FALSE;
   instCmAnodeNgBoxLiftUpDown.statDiagnostics.status := 16#7003;
   instCmAnodeNgBoxLiftUpDown.statDiagnostics.subfunctionStatus := 16#0000;
   instCmAnodeNgBoxLiftUpDown.statDiagnostics.stateNumber := 0;
   instCmAnodeNgBoxLiftUpDown.statEnablePrevious := TRUE;
   instCmAnodeNgBoxLiftUpDown.statFirstCall := FALSE;
   instCmAnodeNgBoxLiftUpDown.statResetPrevious := FALSE;
   instCmAnodeNgBoxLiftUpDown.statValid := TRUE;
   instCmAnodeNgBoxLiftUpDown.statBusy := TRUE;
   instCmAnodeNgBoxLiftUpDown.statError := FALSE;
   instCmAnodeNgBoxLiftUpDown.statInterlockWorkOff := FALSE;
   instCmAnodeNgBoxLiftUpDown.statInterlockHomeOff := FALSE;
   instCmAnodeNgBoxLiftUpDown.statFbState := 50;
   instCmAnodeNgBoxLiftUpDown.statFbStatePrevious := 50;
   instCmAnodeNgBoxLiftUpDown.statErrorUserCleared := FALSE;
   instCmAnodeNgBoxLiftUpDown.statErrorAutoCleared := FALSE;
   instCmAnodeNgBoxLiftUpDown.statErrorState := 16#0000;
   instCmAnodeNgBoxLiftUpDown.statDisablingCompleted := FALSE;
   instCmAnodeNgBoxLiftUpDown.statFeedbackHomePos := TRUE;
   instCmAnodeNgBoxLiftUpDown.statFeedbackWorkPos := FALSE;
   instCmAnodeNgBoxLockUpDown.enable := TRUE;
   instCmAnodeNgBoxLockUpDown.parentReferenceDesignator := WSTRING#'';
   instCmAnodeNgBoxLockUpDown.feedbackHomePos := TRUE;
   instCmAnodeNgBoxLockUpDown.feedbackWorkPos := FALSE;
   instCmAnodeNgBoxLockUpDown.enableManualCmds := TRUE;
   instCmAnodeNgBoxLockUpDown.interlockWorkPos := TRUE;
   instCmAnodeNgBoxLockUpDown.interlockHomePos := TRUE;
   instCmAnodeNgBoxLockUpDown.goToHomePos := FALSE;
   instCmAnodeNgBoxLockUpDown.goToWorkPos := FALSE;
   instCmAnodeNgBoxLockUpDown.statProcessValues.enable := TRUE;
   instCmAnodeNgBoxLockUpDown.statProcessValues.referenceDesignator := WSTRING#'NgBoxLockUpDown';
   instCmAnodeNgBoxLockUpDown.statProcessValues.commandHomePos := FALSE;
   instCmAnodeNgBoxLockUpDown.statProcessValues.commandWorkPos := FALSE;
   instCmAnodeNgBoxLockUpDown.statProcessValues.goToHomePos := FALSE;
   instCmAnodeNgBoxLockUpDown.statProcessValues.goToWorkPos := FALSE;
   instCmAnodeNgBoxLockUpDown.statProcessValues.inHomePos := TRUE;
   instCmAnodeNgBoxLockUpDown.statProcessValues.inWorkPos := FALSE;
   instCmAnodeNgBoxLockUpDown.statProcessValues.reset := FALSE;
   instCmAnodeNgBoxLockUpDown.statProcessValues.enableManualCmds := TRUE;
   instCmAnodeNgBoxLockUpDown.statProcessValues.error := FALSE;
   instCmAnodeNgBoxLockUpDown.statProcessValues.interlockHomePos := TRUE;
   instCmAnodeNgBoxLockUpDown.statProcessValues.interlockWorkPos := TRUE;
   instCmAnodeNgBoxLockUpDown.statProcessValues.status := 16#7003;
   instCmAnodeNgBoxLockUpDown.statProcessValues.interlockWarningWorkPos := FALSE;
   instCmAnodeNgBoxLockUpDown.statProcessValues.interlockWarningHomePos := FALSE;
   instCmAnodeNgBoxLockUpDown.statCurrentInputs.commandHomePos := FALSE;
   instCmAnodeNgBoxLockUpDown.statCurrentInputs.commandWorkPos := FALSE;
   instCmAnodeNgBoxLockUpDown.statCurrentInputs.reset := FALSE;
   instCmAnodeNgBoxLockUpDown.statPreviousInputs.commandHomePos := FALSE;
   instCmAnodeNgBoxLockUpDown.statPreviousInputs.commandWorkPos := FALSE;
   instCmAnodeNgBoxLockUpDown.statPreviousInputs.reset := FALSE;
   instCmAnodeNgBoxLockUpDown.statCurrentInterface.commandHomePos := FALSE;
   instCmAnodeNgBoxLockUpDown.statCurrentInterface.commandWorkPos := FALSE;
   instCmAnodeNgBoxLockUpDown.statCurrentInterface.reset := FALSE;
   instCmAnodeNgBoxLockUpDown.statPreviousInterface.commandHomePos := FALSE;
   instCmAnodeNgBoxLockUpDown.statPreviousInterface.commandWorkPos := FALSE;
   instCmAnodeNgBoxLockUpDown.statPreviousInterface.reset := FALSE;
   instCmAnodeNgBoxLockUpDown.statEmptyDiagnostics.status := 16#0000;
   instCmAnodeNgBoxLockUpDown.statEmptyDiagnostics.subfunctionStatus := 16#0000;
   instCmAnodeNgBoxLockUpDown.statEmptyDiagnostics.stateNumber := 0;
   instCmAnodeNgBoxLockUpDown.instTimerReachPos.PT := T#0MS;
   instCmAnodeNgBoxLockUpDown.instTimerReachPos.IN := FALSE;
   instCmAnodeNgBoxLockUpDown.instTimerLeavePos.PT := T#0MS;
   instCmAnodeNgBoxLockUpDown.instTimerLeavePos.IN := FALSE;
   instCmAnodeNgBoxLockUpDown.instTimerDiscrepancyCheck.PT := T#0MS;
   instCmAnodeNgBoxLockUpDown.instTimerDiscrepancyCheck.IN := FALSE;
   instCmAnodeNgBoxLockUpDown.statDisableAlarms := FALSE;
   instCmAnodeNgBoxLockUpDown.statDiagnostics.status := 16#7003;
   instCmAnodeNgBoxLockUpDown.statDiagnostics.subfunctionStatus := 16#0000;
   instCmAnodeNgBoxLockUpDown.statDiagnostics.stateNumber := 0;
   instCmAnodeNgBoxLockUpDown.statEnablePrevious := TRUE;
   instCmAnodeNgBoxLockUpDown.statFirstCall := FALSE;
   instCmAnodeNgBoxLockUpDown.statResetPrevious := FALSE;
   instCmAnodeNgBoxLockUpDown.statValid := TRUE;
   instCmAnodeNgBoxLockUpDown.statBusy := TRUE;
   instCmAnodeNgBoxLockUpDown.statError := FALSE;
   instCmAnodeNgBoxLockUpDown.statInterlockWorkOff := FALSE;
   instCmAnodeNgBoxLockUpDown.statInterlockHomeOff := FALSE;
   instCmAnodeNgBoxLockUpDown.statFbState := 50;
   instCmAnodeNgBoxLockUpDown.statFbStatePrevious := 50;
   instCmAnodeNgBoxLockUpDown.statErrorUserCleared := FALSE;
   instCmAnodeNgBoxLockUpDown.statErrorAutoCleared := FALSE;
   instCmAnodeNgBoxLockUpDown.statErrorState := 16#0000;
   instCmAnodeNgBoxLockUpDown.statDisablingCompleted := FALSE;
   instCmAnodeNgBoxLockUpDown.statFeedbackHomePos := TRUE;
   instCmAnodeNgBoxLockUpDown.statFeedbackWorkPos := FALSE;
   instCmAnodeNgPnpVaccum.enable := TRUE;
   instCmAnodeNgPnpVaccum.parentReferenceDesignator := WSTRING#'';
   instCmAnodeNgPnpVaccum.feedbackHomePos := TRUE;
   instCmAnodeNgPnpVaccum.feedbackWorkPos := FALSE;
   instCmAnodeNgPnpVaccum.enableManualCmds := TRUE;
   instCmAnodeNgPnpVaccum.interlockWorkPos := TRUE;
   instCmAnodeNgPnpVaccum.interlockHomePos := TRUE;
   instCmAnodeNgPnpVaccum.goToHomePos := FALSE;
   instCmAnodeNgPnpVaccum.goToWorkPos := FALSE;
   instCmAnodeNgPnpVaccum.statProcessValues.enable := TRUE;
   instCmAnodeNgPnpVaccum.statProcessValues.referenceDesignator := WSTRING#'NgPnpVaccum';
   instCmAnodeNgPnpVaccum.statProcessValues.commandHomePos := FALSE;
   instCmAnodeNgPnpVaccum.statProcessValues.commandWorkPos := FALSE;
   instCmAnodeNgPnpVaccum.statProcessValues.goToHomePos := FALSE;
   instCmAnodeNgPnpVaccum.statProcessValues.goToWorkPos := FALSE;
   instCmAnodeNgPnpVaccum.statProcessValues.inHomePos := TRUE;
   instCmAnodeNgPnpVaccum.statProcessValues.inWorkPos := FALSE;
   instCmAnodeNgPnpVaccum.statProcessValues.reset := FALSE;
   instCmAnodeNgPnpVaccum.statProcessValues.enableManualCmds := TRUE;
   instCmAnodeNgPnpVaccum.statProcessValues.error := FALSE;
   instCmAnodeNgPnpVaccum.statProcessValues.interlockHomePos := TRUE;
   instCmAnodeNgPnpVaccum.statProcessValues.interlockWorkPos := TRUE;
   instCmAnodeNgPnpVaccum.statProcessValues.status := 16#7003;
   instCmAnodeNgPnpVaccum.statProcessValues.interlockWarningWorkPos := FALSE;
   instCmAnodeNgPnpVaccum.statProcessValues.interlockWarningHomePos := FALSE;
   instCmAnodeNgPnpVaccum.statCurrentInputs.commandHomePos := FALSE;
   instCmAnodeNgPnpVaccum.statCurrentInputs.commandWorkPos := FALSE;
   instCmAnodeNgPnpVaccum.statCurrentInputs.reset := FALSE;
   instCmAnodeNgPnpVaccum.statPreviousInputs.commandHomePos := FALSE;
   instCmAnodeNgPnpVaccum.statPreviousInputs.commandWorkPos := FALSE;
   instCmAnodeNgPnpVaccum.statPreviousInputs.reset := FALSE;
   instCmAnodeNgPnpVaccum.statCurrentInterface.commandHomePos := FALSE;
   instCmAnodeNgPnpVaccum.statCurrentInterface.commandWorkPos := FALSE;
   instCmAnodeNgPnpVaccum.statCurrentInterface.reset := FALSE;
   instCmAnodeNgPnpVaccum.statPreviousInterface.commandHomePos := FALSE;
   instCmAnodeNgPnpVaccum.statPreviousInterface.commandWorkPos := FALSE;
   instCmAnodeNgPnpVaccum.statPreviousInterface.reset := FALSE;
   instCmAnodeNgPnpVaccum.statEmptyDiagnostics.status := 16#0000;
   instCmAnodeNgPnpVaccum.statEmptyDiagnostics.subfunctionStatus := 16#0000;
   instCmAnodeNgPnpVaccum.statEmptyDiagnostics.stateNumber := 0;
   instCmAnodeNgPnpVaccum.instTimerReachPos.PT := T#0MS;
   instCmAnodeNgPnpVaccum.instTimerReachPos.IN := FALSE;
   instCmAnodeNgPnpVaccum.instTimerLeavePos.PT := T#0MS;
   instCmAnodeNgPnpVaccum.instTimerLeavePos.IN := FALSE;
   instCmAnodeNgPnpVaccum.instTimerDiscrepancyCheck.PT := T#0MS;
   instCmAnodeNgPnpVaccum.instTimerDiscrepancyCheck.IN := FALSE;
   instCmAnodeNgPnpVaccum.statDisableAlarms := FALSE;
   instCmAnodeNgPnpVaccum.statDiagnostics.status := 16#7003;
   instCmAnodeNgPnpVaccum.statDiagnostics.subfunctionStatus := 16#0000;
   instCmAnodeNgPnpVaccum.statDiagnostics.stateNumber := 0;
   instCmAnodeNgPnpVaccum.statEnablePrevious := TRUE;
   instCmAnodeNgPnpVaccum.statFirstCall := FALSE;
   instCmAnodeNgPnpVaccum.statResetPrevious := FALSE;
   instCmAnodeNgPnpVaccum.statValid := TRUE;
   instCmAnodeNgPnpVaccum.statBusy := TRUE;
   instCmAnodeNgPnpVaccum.statError := FALSE;
   instCmAnodeNgPnpVaccum.statInterlockWorkOff := FALSE;
   instCmAnodeNgPnpVaccum.statInterlockHomeOff := FALSE;
   instCmAnodeNgPnpVaccum.statFbState := 50;
   instCmAnodeNgPnpVaccum.statFbStatePrevious := 50;
   instCmAnodeNgPnpVaccum.statErrorUserCleared := FALSE;
   instCmAnodeNgPnpVaccum.statErrorAutoCleared := FALSE;
   instCmAnodeNgPnpVaccum.statErrorState := 16#0000;
   instCmAnodeNgPnpVaccum.statDisablingCompleted := FALSE;
   instCmAnodeNgPnpVaccum.statFeedbackHomePos := TRUE;
   instCmAnodeNgPnpVaccum.statFeedbackWorkPos := FALSE;
   instCmAnodeConveyorCoverFwdBwd.enable := TRUE;
   instCmAnodeConveyorCoverFwdBwd.parentReferenceDesignator := WSTRING#'';
   instCmAnodeConveyorCoverFwdBwd.feedbackHomePos := FALSE;
   instCmAnodeConveyorCoverFwdBwd.feedbackWorkPos := FALSE;
   instCmAnodeConveyorCoverFwdBwd.enableManualCmds := TRUE;
   instCmAnodeConveyorCoverFwdBwd.interlockWorkPos := TRUE;
   instCmAnodeConveyorCoverFwdBwd.interlockHomePos := TRUE;
   instCmAnodeConveyorCoverFwdBwd.goToHomePos := FALSE;
   instCmAnodeConveyorCoverFwdBwd.goToWorkPos := FALSE;
   instCmAnodeConveyorCoverFwdBwd.statProcessValues.enable := TRUE;
   instCmAnodeConveyorCoverFwdBwd.statProcessValues.referenceDesignator := WSTRING#'ConveyorCoverFwdBwd';
   instCmAnodeConveyorCoverFwdBwd.statProcessValues.commandHomePos := FALSE;
   instCmAnodeConveyorCoverFwdBwd.statProcessValues.commandWorkPos := FALSE;
   instCmAnodeConveyorCoverFwdBwd.statProcessValues.goToHomePos := FALSE;
   instCmAnodeConveyorCoverFwdBwd.statProcessValues.goToWorkPos := FALSE;
   instCmAnodeConveyorCoverFwdBwd.statProcessValues.inHomePos := FALSE;
   instCmAnodeConveyorCoverFwdBwd.statProcessValues.inWorkPos := FALSE;
   instCmAnodeConveyorCoverFwdBwd.statProcessValues.reset := FALSE;
   instCmAnodeConveyorCoverFwdBwd.statProcessValues.enableManualCmds := TRUE;
   instCmAnodeConveyorCoverFwdBwd.statProcessValues.error := FALSE;
   instCmAnodeConveyorCoverFwdBwd.statProcessValues.interlockHomePos := TRUE;
   instCmAnodeConveyorCoverFwdBwd.statProcessValues.interlockWorkPos := TRUE;
   instCmAnodeConveyorCoverFwdBwd.statProcessValues.status := 16#7003;
   instCmAnodeConveyorCoverFwdBwd.statProcessValues.interlockWarningWorkPos := FALSE;
   instCmAnodeConveyorCoverFwdBwd.statProcessValues.interlockWarningHomePos := FALSE;
   instCmAnodeConveyorCoverFwdBwd.statCurrentInputs.commandHomePos := FALSE;
   instCmAnodeConveyorCoverFwdBwd.statCurrentInputs.commandWorkPos := FALSE;
   instCmAnodeConveyorCoverFwdBwd.statCurrentInputs.reset := FALSE;
   instCmAnodeConveyorCoverFwdBwd.statPreviousInputs.commandHomePos := FALSE;
   instCmAnodeConveyorCoverFwdBwd.statPreviousInputs.commandWorkPos := FALSE;
   instCmAnodeConveyorCoverFwdBwd.statPreviousInputs.reset := FALSE;
   instCmAnodeConveyorCoverFwdBwd.statCurrentInterface.commandHomePos := FALSE;
   instCmAnodeConveyorCoverFwdBwd.statCurrentInterface.commandWorkPos := FALSE;
   instCmAnodeConveyorCoverFwdBwd.statCurrentInterface.reset := FALSE;
   instCmAnodeConveyorCoverFwdBwd.statPreviousInterface.commandHomePos := FALSE;
   instCmAnodeConveyorCoverFwdBwd.statPreviousInterface.commandWorkPos := FALSE;
   instCmAnodeConveyorCoverFwdBwd.statPreviousInterface.reset := FALSE;
   instCmAnodeConveyorCoverFwdBwd.statEmptyDiagnostics.status := 16#0000;
   instCmAnodeConveyorCoverFwdBwd.statEmptyDiagnostics.subfunctionStatus := 16#0000;
   instCmAnodeConveyorCoverFwdBwd.statEmptyDiagnostics.stateNumber := 0;
   instCmAnodeConveyorCoverFwdBwd.instTimerReachPos.PT := T#0MS;
   instCmAnodeConveyorCoverFwdBwd.instTimerReachPos.IN := FALSE;
   instCmAnodeConveyorCoverFwdBwd.instTimerLeavePos.PT := T#0MS;
   instCmAnodeConveyorCoverFwdBwd.instTimerLeavePos.IN := FALSE;
   instCmAnodeConveyorCoverFwdBwd.instTimerDiscrepancyCheck.PT := T#0MS;
   instCmAnodeConveyorCoverFwdBwd.instTimerDiscrepancyCheck.IN := FALSE;
   instCmAnodeConveyorCoverFwdBwd.statDisableAlarms := FALSE;
   instCmAnodeConveyorCoverFwdBwd.statDiagnostics.status := 16#7003;
   instCmAnodeConveyorCoverFwdBwd.statDiagnostics.subfunctionStatus := 16#0000;
   instCmAnodeConveyorCoverFwdBwd.statDiagnostics.stateNumber := 0;
   instCmAnodeConveyorCoverFwdBwd.statEnablePrevious := TRUE;
   instCmAnodeConveyorCoverFwdBwd.statFirstCall := FALSE;
   instCmAnodeConveyorCoverFwdBwd.statResetPrevious := FALSE;
   instCmAnodeConveyorCoverFwdBwd.statValid := TRUE;
   instCmAnodeConveyorCoverFwdBwd.statBusy := TRUE;
   instCmAnodeConveyorCoverFwdBwd.statError := FALSE;
   instCmAnodeConveyorCoverFwdBwd.statInterlockWorkOff := FALSE;
   instCmAnodeConveyorCoverFwdBwd.statInterlockHomeOff := FALSE;
   instCmAnodeConveyorCoverFwdBwd.statFbState := 50;
   instCmAnodeConveyorCoverFwdBwd.statFbStatePrevious := 50;
   instCmAnodeConveyorCoverFwdBwd.statErrorUserCleared := FALSE;
   instCmAnodeConveyorCoverFwdBwd.statErrorAutoCleared := FALSE;
   instCmAnodeConveyorCoverFwdBwd.statErrorState := 16#0000;
   instCmAnodeConveyorCoverFwdBwd.statDisablingCompleted := FALSE;
   instCmAnodeConveyorCoverFwdBwd.statFeedbackHomePos := FALSE;
   instCmAnodeConveyorCoverFwdBwd.statFeedbackWorkPos := FALSE;
   instCmAnodeConveyorPickUpBlower.enable := TRUE;
   instCmAnodeConveyorPickUpBlower.parentReferenceDesignator := WSTRING#'';
   instCmAnodeConveyorPickUpBlower.feedbackHomePos := FALSE;
   instCmAnodeConveyorPickUpBlower.feedbackWorkPos := FALSE;
   instCmAnodeConveyorPickUpBlower.enableManualCmds := TRUE;
   instCmAnodeConveyorPickUpBlower.interlockWorkPos := TRUE;
   instCmAnodeConveyorPickUpBlower.interlockHomePos := TRUE;
   instCmAnodeConveyorPickUpBlower.goToHomePos := FALSE;
   instCmAnodeConveyorPickUpBlower.goToWorkPos := FALSE;
   instCmAnodeConveyorPickUpBlower.statProcessValues.enable := TRUE;
   instCmAnodeConveyorPickUpBlower.statProcessValues.referenceDesignator := WSTRING#'ConveyorPickUpBlower';
   instCmAnodeConveyorPickUpBlower.statProcessValues.commandHomePos := FALSE;
   instCmAnodeConveyorPickUpBlower.statProcessValues.commandWorkPos := FALSE;
   instCmAnodeConveyorPickUpBlower.statProcessValues.goToHomePos := FALSE;
   instCmAnodeConveyorPickUpBlower.statProcessValues.goToWorkPos := FALSE;
   instCmAnodeConveyorPickUpBlower.statProcessValues.inHomePos := FALSE;
   instCmAnodeConveyorPickUpBlower.statProcessValues.inWorkPos := FALSE;
   instCmAnodeConveyorPickUpBlower.statProcessValues.reset := FALSE;
   instCmAnodeConveyorPickUpBlower.statProcessValues.enableManualCmds := TRUE;
   instCmAnodeConveyorPickUpBlower.statProcessValues.error := FALSE;
   instCmAnodeConveyorPickUpBlower.statProcessValues.interlockHomePos := TRUE;
   instCmAnodeConveyorPickUpBlower.statProcessValues.interlockWorkPos := TRUE;
   instCmAnodeConveyorPickUpBlower.statProcessValues.status := 16#7003;
   instCmAnodeConveyorPickUpBlower.statProcessValues.interlockWarningWorkPos := FALSE;
   instCmAnodeConveyorPickUpBlower.statProcessValues.interlockWarningHomePos := FALSE;
   instCmAnodeConveyorPickUpBlower.statCurrentInputs.commandHomePos := FALSE;
   instCmAnodeConveyorPickUpBlower.statCurrentInputs.commandWorkPos := FALSE;
   instCmAnodeConveyorPickUpBlower.statCurrentInputs.reset := FALSE;
   instCmAnodeConveyorPickUpBlower.statPreviousInputs.commandHomePos := FALSE;
   instCmAnodeConveyorPickUpBlower.statPreviousInputs.commandWorkPos := FALSE;
   instCmAnodeConveyorPickUpBlower.statPreviousInputs.reset := FALSE;
   instCmAnodeConveyorPickUpBlower.statCurrentInterface.commandHomePos := FALSE;
   instCmAnodeConveyorPickUpBlower.statCurrentInterface.commandWorkPos := FALSE;
   instCmAnodeConveyorPickUpBlower.statCurrentInterface.reset := FALSE;
   instCmAnodeConveyorPickUpBlower.statPreviousInterface.commandHomePos := FALSE;
   instCmAnodeConveyorPickUpBlower.statPreviousInterface.commandWorkPos := FALSE;
   instCmAnodeConveyorPickUpBlower.statPreviousInterface.reset := FALSE;
   instCmAnodeConveyorPickUpBlower.statEmptyDiagnostics.status := 16#0000;
   instCmAnodeConveyorPickUpBlower.statEmptyDiagnostics.subfunctionStatus := 16#0000;
   instCmAnodeConveyorPickUpBlower.statEmptyDiagnostics.stateNumber := 0;
   instCmAnodeConveyorPickUpBlower.instTimerReachPos.PT := T#0MS;
   instCmAnodeConveyorPickUpBlower.instTimerReachPos.IN := FALSE;
   instCmAnodeConveyorPickUpBlower.instTimerLeavePos.PT := T#0MS;
   instCmAnodeConveyorPickUpBlower.instTimerLeavePos.IN := FALSE;
   instCmAnodeConveyorPickUpBlower.instTimerDiscrepancyCheck.PT := T#0MS;
   instCmAnodeConveyorPickUpBlower.instTimerDiscrepancyCheck.IN := FALSE;
   instCmAnodeConveyorPickUpBlower.statDisableAlarms := FALSE;
   instCmAnodeConveyorPickUpBlower.statDiagnostics.status := 16#7003;
   instCmAnodeConveyorPickUpBlower.statDiagnostics.subfunctionStatus := 16#0000;
   instCmAnodeConveyorPickUpBlower.statDiagnostics.stateNumber := 0;
   instCmAnodeConveyorPickUpBlower.statEnablePrevious := TRUE;
   instCmAnodeConveyorPickUpBlower.statFirstCall := FALSE;
   instCmAnodeConveyorPickUpBlower.statResetPrevious := FALSE;
   instCmAnodeConveyorPickUpBlower.statValid := TRUE;
   instCmAnodeConveyorPickUpBlower.statBusy := TRUE;
   instCmAnodeConveyorPickUpBlower.statError := FALSE;
   instCmAnodeConveyorPickUpBlower.statInterlockWorkOff := FALSE;
   instCmAnodeConveyorPickUpBlower.statInterlockHomeOff := FALSE;
   instCmAnodeConveyorPickUpBlower.statFbState := 50;
   instCmAnodeConveyorPickUpBlower.statFbStatePrevious := 50;
   instCmAnodeConveyorPickUpBlower.statErrorUserCleared := FALSE;
   instCmAnodeConveyorPickUpBlower.statErrorAutoCleared := FALSE;
   instCmAnodeConveyorPickUpBlower.statErrorState := 16#0000;
   instCmAnodeConveyorPickUpBlower.statDisablingCompleted := FALSE;
   instCmAnodeConveyorPickUpBlower.statFeedbackHomePos := FALSE;
   instCmAnodeConveyorPickUpBlower.statFeedbackWorkPos := FALSE;
   instManageAlarms.proDiagState.Total_Number := 500;
   instManageAlarms.proDiagState.All := TRUE;
   instManageAlarms.proDiagState.O := FALSE;
   instManageAlarms.proDiagState.I := FALSE;
   instManageAlarms.proDiagState.R := FALSE;
   instManageAlarms.proDiagState."A" := FALSE;
   instManageAlarms.proDiagState.P := FALSE;
   instManageAlarms.proDiagState.Merr := TRUE;
   instManageAlarms.proDiagState.Mtxt := FALSE;
   instManageAlarms.proDiagState.SV_Types := 16#20;
   instManageAlarms.proDiagState.C1 := TRUE;
   instManageAlarms.proDiagState.C2 := FALSE;
   instManageAlarms.proDiagState.C3 := FALSE;
   instManageAlarms.proDiagState.C4 := FALSE;
   instManageAlarms.proDiagState.C5 := FALSE;
   instManageAlarms.proDiagState.C6 := FALSE;
   instManageAlarms.proDiagState.C7 := FALSE;
   instManageAlarms.proDiagState.C8 := FALSE;
   instManageAlarms.proDiagState.Categories := 16#01;
   instManageAlarms.proDiagState.Sub_Cat_1 := 16#0000_0001;
   instManageAlarms.proDiagState.Sub_Cat_2 := 16#0000_0000;
   instManageAlarms.proDiagState.Reserved := 16#00;
   instManageAlarms.parentAlarmDB.error := TRUE;
   instManageAlarms.parentAlarmDB.warning := FALSE;
   instManageAlarms.parentAlarmDB.info := FALSE;
   instManageAlarms.alarmDB.error := TRUE;
   instManageAlarms.alarmDB.warning := FALSE;
   instManageAlarms.alarmDB.info := FALSE;
   instManageAlarms.hmiInterfaceDB.error := TRUE;
   instManageAlarms.hmiInterfaceDB.warning := FALSE;
   instManageAlarms.hmiInterfaceDB.info := FALSE;
   statUnitStatus.acknowledgeActive := FALSE;
   statUnitStatus.alarmsDisabled := FALSE;
   statUnitStatus.simulationActive := FALSE;
   statUnitStatus.safetyReleased := TRUE;
   statUnitStatus.specialFunctions.GaugeRnR1AnodeAlign := FALSE;
   statUnitStatus.specialFunctions.GaugeRnR1CathodeAlign := FALSE;
   statUnitStatus.specialFunctions.GaugeRnR3AnodeAlign := FALSE;
   statUnitStatus.specialFunctions.GaugeRnR3CathodeAlign := FALSE;
   statUnitStatus.specialFunctions.releaseEntry := FALSE;
   statUnitStatus.specialFunctions.dryRun := FALSE;
   statUnitStatus.specialFunctions.ReelCutAnodeUnuse := FALSE;
   statUnitStatus.mode.current := 2;
   statUnitStatus.mode.production := FALSE;
   statUnitStatus.mode.maintenance := TRUE;
   statUnitStatus.mode.manual := FALSE;
   statUnitStatus.mode.sleep := FALSE;
   statUnitStatus.mode.deepsleep := FALSE;
   statUnitStatus.mode.userMode04 := FALSE;
   statUnitStatus.mode.userMode05 := FALSE;
   statUnitStatus.mode.userMode06 := FALSE;
   statUnitStatus.mode.userMode07 := FALSE;
   statUnitStatus.mode.userMode08 := FALSE;
   statUnitStatus.mode.userMode09 := FALSE;
   statUnitStatus.mode.userMode10 := FALSE;
   statUnitStatus.mode.userMode11 := FALSE;
   statUnitStatus.mode.userMode12 := FALSE;
   statUnitStatus.mode.userMode13 := FALSE;
   statUnitStatus.state.current := 2;
   statUnitStatus.state.clearing := FALSE;
   statUnitStatus.state.stopped := TRUE;
   statUnitStatus.state.starting := FALSE;
   statUnitStatus.state.idle := FALSE;
   statUnitStatus.state.suspended := FALSE;
   statUnitStatus.state.execute := FALSE;
   statUnitStatus.state.stopping := FALSE;
   statUnitStatus.state.aborting := FALSE;
   statUnitStatus.state.aborted := FALSE;
   statUnitStatus.state.holding := FALSE;
   statUnitStatus.state.held := FALSE;
   statUnitStatus.state.unholding := FALSE;
   statUnitStatus.state.suspending := FALSE;
   statUnitStatus.state.unsuspending := FALSE;
   statUnitStatus.state.resetting := FALSE;
   statUnitStatus.state.completing := FALSE;
   statUnitStatus.state.complete := FALSE;
END_DATA_BLOCK
